LIN {X 0,Y 524.176,Z 655.147,A -85,B 0,C 180,E1 -4756.825,E2 -4756.825} C_VEL
LIN {X 0,Y 523.934,Z 664.266,A -85,B 0,C 180,E1 -4758.392,E2 -4758.392} C_VEL
LIN {X 0,Y 523.658,Z 671.855,A -85,B 0,C 180,E1 -4759.952,E2 -4759.952} C_VEL
LIN {X 0,Y 523.503,Z 679.465,A -85,B 0,C 180,E1 -4761.897,E2 -4761.897} C_VEL
LIN {X 0,Y 523.41,Z 685.25,A -85,B 0,C 180,E1 -4763.834,E2 -4763.834} C_VEL
LIN {X 0,Y 523.312,Z 688.633,A -85,B 0,C 180,E1 -4765.378,E2 -4765.378} C_VEL
LIN {X 0,Y 523.353,Z 691.091,A -85,B 0,C 180,E1 -4766.921,E2 -4766.921} C_VEL
LIN {X 0,Y 523.268,Z 692.478,A -85,B 0,C 180,E1 -4768.461,E2 -4768.461} C_VEL
LIN {X 0,Y 523.242,Z 693,A -85,B 0,C 180,E1 -4770,E2 -4770} C_VEL
LIN {X 0,Y 523.268,Z 692.477,A -85,B 0,C 180,E1 -4771.539,E2 -4771.539} C_VEL
LIN {X 0,Y 523.353,Z 691.089,A -85,B 0,C 180,E1 -4773.079,E2 -4773.079} C_VEL
LIN {X 0,Y 523.312,Z 688.633,A -85,B 0,C 180,E1 -4774.622,E2 -4774.622} C_VEL
LIN {X 0,Y 523.41,Z 685.253,A -85,B 0,C 180,E1 -4776.167,E2 -4776.167} C_VEL
LIN {X 0,Y 523.503,Z 679.467,A -85,B 0,C 180,E1 -4778.104,E2 -4778.104} C_VEL
LIN {X 0,Y 523.658,Z 671.854,A -85,B 0,C 180,E1 -4780.048,E2 -4780.048} C_VEL
LIN {X 0,Y 523.956,Z 663.711,A -85,B 0,C 180,E1 -4781.715,E2 -4781.715} C_VEL
LIN {X 0,Y 524.176,Z 655.145,A -85,B 0,C 180,E1 -4783.175,E2 -4783.175} C_VEL
LIN {X 0,Y 524.649,Z 644.262,A -85,B 0,C 180,E1 -4784.745,E2 -4784.745} C_VEL
LIN {X 0,Y 525.099,Z 633.027,A -85,B 0,C 180,E1 -4786.124,E2 -4786.124} C_VEL
LIN {X 0,Y 525.666,Z 620.786,A -85,B 0,C 180,E1 -4787.406,E2 -4787.406} C_VEL
LIN {X 0,Y 526.239,Z 607.333,A -85,B 0,C 180,E1 -4788.601,E2 -4788.601} C_VEL
LIN {X 0,Y 526.827,Z 594.297,A -85,B 0,C 180,E1 -4789.583,E2 -4789.583} C_VEL
LIN {X 0,Y 527.381,Z 580.397,A -85,B 0,C 180,E1 -4790.476,E2 -4790.476} C_VEL
LIN {X 0,Y 528.118,Z 564.128,A -85,B 0,C 180,E1 -4791.326,E2 -4791.326} C_VEL
LIN {X 0,Y 528.555,Z 550.131,A -85,B 0,C 180,E1 -4791.909,E2 -4791.909} C_VEL
LIN {X 0,Y 529.007,Z 533.263,A -85,B 0,C 180,E1 -4792.455,E2 -4792.455} C_VEL
LIN {X 0,Y 529.386,Z 516.858,A -85,B 0,C 180,E1 -4792.824,E2 -4792.824} C_VEL
LIN {X 0,Y 530.879,Z 326.095,A -85,B 0,C 180,E1 -4795.547,E2 -4795.547} C_VEL
LIN {X 0,Y 528.167,Z 310.802,A -85,B 0,C 180,E1 -4795.922,E2 -4795.922} C_VEL
LIN {X 0,Y 529.041,Z 286.938,A -85,B 0,C 180,E1 -4798.168,E2 -4798.168} C_VEL
LIN {X 0,Y 523.929,Z 269.536,A -85,B 0,C 180,E1 -4800.201,E2 -4800.201} C_VEL
LIN {X 0,Y 523.94,Z 269.535,A -85,B 0,C 180,E1 -4803.365,E2 -4803.365} C_VEL
LIN {X 0,Y 523.902,Z 269.536,A -85,B 0,C 180,E1 -4806.402,E2 -4806.402} C_VEL
LIN {X 0,Y 523.922,Z 269.536,A -85,B 0,C 180,E1 -4809.085,E2 -4809.085} C_VEL
LIN {X 0,Y 523.957,Z 269.524,A -85,B 0,C 180,E1 -4812.119,E2 -4812.119} C_VEL
LIN {X 0,Y 523.956,Z 269.53,A -85,B 0,C 180,E1 -4815.309,E2 -4815.309} C_VEL
LIN {X 0,Y 523.962,Z 269.527,A -85,B 0,C 180,E1 -4818.689,E2 -4818.689} C_VEL
LIN {X 0,Y 523.917,Z 269.529,A -85,B 0,C 180,E1 -4821.899,E2 -4821.899} C_VEL
LIN {X 0,Y 523.925,Z 269.539,A -85,B 0,C 180,E1 -4824.911,E2 -4824.911} C_VEL
LIN {X 0,Y 523.936,Z 269.527,A -85,B 0,C 180,E1 -4827.68,E2 -4827.68} C_VEL
LIN {X 0,Y 523.955,Z 269.532,A -85,B 0,C 180,E1 -4830.677,E2 -4830.677} C_VEL
LIN {X 0,Y 523.975,Z 269.524,A -85,B 0,C 180,E1 -4833.729,E2 -4833.729} C_VEL
LIN {X 0,Y 523.937,Z 269.53,A -85,B 0,C 180,E1 -4836.271,E2 -4836.271} C_VEL
LIN {X 0,Y 523.947,Z 269.531,A -85,B 0,C 180,E1 -4838.767,E2 -4838.767} C_VEL
LIN {X 0,Y 523.95,Z 269.528,A -85,B 0,C 180,E1 -4841.221,E2 -4841.221} C_VEL
LIN {X 0,Y 523.932,Z 269.522,A -85,B 0,C 180,E1 -4843.639,E2 -4843.639} C_VEL
LIN {X 0,Y 523.934,Z 269.531,A -85,B 0,C 180,E1 -4846.028,E2 -4846.028} C_VEL
LIN {X 0,Y 524.015,Z 269.521,A -85,B 0,C 180,E1 -4848.395,E2 -4848.395} C_VEL
LIN {X 0,Y 523.988,Z 269.522,A -85,B 0,C 180,E1 -4851.516,E2 -4851.516} C_VEL
LIN {X 0,Y 524.069,Z 269.511,A -85,B 0,C 180,E1 -4854.614,E2 -4854.614} C_VEL
LIN {X 0,Y 524.111,Z 269.506,A -85,B 0,C 180,E1 -4857.695,E2 -4857.695} C_VEL
LIN {X 0,Y 524.121,Z 269.503,A -85,B 0,C 180,E1 -4860.769,E2 -4860.769} C_VEL
LIN {X 0,Y 524.006,Z 269.519,A -85,B 0,C 180,E1 -4863.076,E2 -4863.076} C_VEL
LIN {X 0,Y 524.066,Z 269.513,A -85,B 0,C 180,E1 -4865.387,E2 -4865.387} C_VEL
LIN {X 0,Y 523.957,Z 269.526,A -85,B 0,C 180,E1 -4868.485,E2 -4868.485} C_VEL
LIN {X 0,Y 524.002,Z 269.523,A -85,B 0,C 180,E1 -4871.737,E2 -4871.737} C_VEL
LIN {X 0,Y 523.99,Z 269.521,A -85,B 0,C 180,E1 -4875.05,E2 -4875.05} C_VEL
LIN {X 0,Y 523.917,Z 269.537,A -85,B 0,C 180,E1 -4877.971,E2 -4877.971} C_VEL
LIN {X 0,Y 523.952,Z 269.533,A -85,B 0,C 180,E1 -4880.411,E2 -4880.411} C_VEL
LIN {X 0,Y 523.903,Z 269.531,A -85,B 0,C 180,E1 -4882.894,E2 -4882.894} C_VEL
LIN {X 0,Y 523.879,Z 269.536,A -85,B 0,C 180,E1 -4885.423,E2 -4885.423} C_VEL
LIN {X 0,Y 523.897,Z 269.536,A -85,B 0,C 180,E1 -4888.004,E2 -4888.004} C_VEL
LIN {X 0,Y 523.901,Z 269.534,A -85,B 0,C 180,E1 -4890.846,E2 -4890.846} C_VEL
LIN {X 0,Y 523.914,Z 269.538,A -85,B 0,C 180,E1 -4893.727,E2 -4893.727} C_VEL
LIN {X 0,Y 523.85,Z 269.546,A -85,B 0,C 180,E1 -4896.393,E2 -4896.393} C_VEL
LIN {X 0,Y 523.894,Z 269.535,A -85,B 0,C 180,E1 -4899.088,E2 -4899.088} C_VEL
LIN {X 0,Y 523.889,Z 269.542,A -85,B 0,C 180,E1 -4902.126,E2 -4902.126} C_VEL
LIN {X 0,Y 523.935,Z 269.533,A -85,B 0,C 180,E1 -4905.312,E2 -4905.312} C_VEL
LIN {X 0,Y 523.878,Z 269.537,A -85,B 0,C 180,E1 -4906.903,E2 -4906.903} C_VEL
LIN {X 0,Y 523.085,Z 269.695,A -85,B 0,C 180,E1 -4907.359,E2 -4907.359} C_VEL
LIN {X 0,Y 517.322,Z 270.465,A -85,B 0,C 180,E1 -4908.74,E2 -4908.74} C_VEL
LIN {X 0,Y 517.059,Z 271.408,A -85,B 0,C 180,E1 -4909.06,E2 -4909.06} C_VEL
LIN {X 0,Y 517.156,Z 271.75,A -85,B 0,C 180,E1 -4909.114,E2 -4909.114} C_VEL
LIN {X 0,Y 520.813,Z 284.323,A -85,B 0,C 180,E1 -4910.753,E2 -4910.753} C_VEL
LIN {X 0,Y 522.606,Z 289.121,A -85,B 0,C 180,E1 -4910.923,E2 -4910.923} C_VEL
LIN {X 0,Y 524.602,Z 299.005,A -85,B 0,C 180,E1 -4911.178,E2 -4911.178} C_VEL
LIN {X 0,Y 522.859,Z 490.272,A -85,B 0,C 180,E1 -4913.95,E2 -4913.95} C_VEL
LIN {X 0,Y 522.455,Z 507.382,A -85,B 0,C 180,E1 -4914.364,E2 -4914.364} C_VEL
LIN {X 0,Y 521.966,Z 523.592,A -85,B 0,C 180,E1 -4914.92,E2 -4914.92} C_VEL
LIN {X 0,Y 521.376,Z 539.542,A -85,B 0,C 180,E1 -4915.635,E2 -4915.635} C_VEL
LIN {X 0,Y 520.708,Z 554.605,A -85,B 0,C 180,E1 -4916.475,E2 -4916.475} C_VEL
LIN {X 0,Y 520.002,Z 569.721,A -85,B 0,C 180,E1 -4917.504,E2 -4917.504} C_VEL
LIN {X 0,Y 519.333,Z 583.007,A -85,B 0,C 180,E1 -4918.59,E2 -4918.59} C_VEL
LIN {X 0,Y 518.659,Z 595.537,A -85,B 0,C 180,E1 -4919.797,E2 -4919.797} C_VEL
LIN {X 0,Y 518.053,Z 607.991,A -85,B 0,C 180,E1 -4921.21,E2 -4921.21} C_VEL
LIN {X 0,Y 517.516,Z 619.257,A -85,B 0,C 180,E1 -4922.72,E2 -4922.72} C_VEL
LIN {X 0,Y 517.107,Z 628.765,A -85,B 0,C 180,E1 -4924.22,E2 -4924.22} C_VEL
LIN {X 0,Y 516.772,Z 637.779,A -85,B 0,C 180,E1 -4925.921,E2 -4925.921} C_VEL
LIN {X 0,Y 516.508,Z 645.511,A -85,B 0,C 180,E1 -4927.709,E2 -4927.709} C_VEL
LIN {X 0,Y 516.4,Z 650.992,A -85,B 0,C 180,E1 -4929.277,E2 -4929.277} C_VEL
LIN {X 0,Y 516.251,Z 655.643,A -85,B 0,C 180,E1 -4930.93,E2 -4930.93} C_VEL
LIN {X 0,Y 516.21,Z 659.042,A -85,B 0,C 180,E1 -4932.571,E2 -4932.571} C_VEL
LIN {X 0,Y 516.137,Z 661.375,A -85,B 0,C 180,E1 -4934.197,E2 -4934.197} C_VEL
LIN {X 0,Y 516.177,Z 662.678,A -85,B 0,C 180,E1 -4935.813,E2 -4935.813} C_VEL
LIN {X 0,Y 516.178,Z 662.93,A -85,B 0,C 180,E1 -4937.417,E2 -4937.417} C_VEL
LIN {X 0,Y 516.258,Z 662.227,A -85,B 0,C 180,E1 -4939.013,E2 -4939.013} C_VEL
LIN {X 0,Y 516.163,Z 660.484,A -85,B 0,C 180,E1 -4940.596,E2 -4940.596} C_VEL
LIN {X 0,Y 516.227,Z 657.838,A -85,B 0,C 180,E1 -4942.175,E2 -4942.175} C_VEL
LIN {X 0,Y 516.391,Z 653.034,A -85,B 0,C 180,E1 -4944.141,E2 -4944.141} C_VEL
LIN {X 0,Y 516.455,Z 647.983,A -85,B 0,C 180,E1 -4945.708,E2 -4945.708} C_VEL
LIN {X 0,Y 516.589,Z 641.868,A -85,B 0,C 180,E1 -4947.271,E2 -4947.271} C_VEL
LIN {X 0,Y 516.908,Z 633.446,A -85,B 0,C 180,E1 -4949.026,E2 -4949.026} C_VEL
LIN {X 0,Y 517.182,Z 624.422,A -85,B 0,C 180,E1 -4950.584,E2 -4950.584} C_VEL
LIN {X 0,Y 517.716,Z 613.744,A -85,B 0,C 180,E1 -4952.139,E2 -4952.139} C_VEL
LIN {X 0,Y 518.308,Z 602.777,A -85,B 0,C 180,E1 -4953.498,E2 -4953.498} C_VEL
LIN {X 0,Y 518.905,Z 590.953,A -85,B 0,C 180,E1 -4954.758,E2 -4954.758} C_VEL
LIN {X 0,Y 519.574,Z 578.074,A -85,B 0,C 180,E1 -4955.92,E2 -4955.92} C_VEL
LIN {X 0,Y 520.204,Z 564.159,A -85,B 0,C 180,E1 -4956.984,E2 -4956.984} C_VEL
LIN {X 0,Y 520.902,Z 548.964,A -85,B 0,C 180,E1 -4957.949,E2 -4957.949} C_VEL
LIN {X 0,Y 521.584,Z 534.106,A -85,B 0,C 180,E1 -4958.719,E2 -4958.719} C_VEL
LIN {X 0,Y 522.114,Z 519.014,A -85,B 0,C 180,E1 -4959.344,E2 -4959.344} C_VEL
LIN {X 0,Y 522.584,Z 502.822,A -85,B 0,C 180,E1 -4959.849,E2 -4959.849} C_VEL
LIN {X 0,Y 522.925,Z 485.838,A -85,B 0,C 180,E1 -4960.213,E2 -4960.213} C_VEL
LIN {X 0,Y 524.588,Z 299.14,A -85,B 0,C 180,E1 -4962.908,E2 -4962.908} C_VEL
LIN {X 0,Y 521.958,Z 287.007,A -85,B 0,C 180,E1 -4963.232,E2 -4963.232} C_VEL
LIN {X 0,Y 520.663,Z 283.932,A -85,B 0,C 180,E1 -4963.375,E2 -4963.375} C_VEL
LIN {X 0,Y 516.944,Z 270.406,A -85,B 0,C 180,E1 -4965.144,E2 -4965.144} C_VEL
LIN {X 0,Y 516.88,Z 270.415,A -85,B 0,C 180,E1 -4968.224,E2 -4968.224} C_VEL
LIN {X 0,Y 516.903,Z 270.41,A -85,B 0,C 180,E1 -4970.702,E2 -4970.702} C_VEL
LIN {X 0,Y 516.86,Z 270.413,A -85,B 0,C 180,E1 -4973.224,E2 -4973.224} C_VEL
LIN {X 0,Y 516.863,Z 270.412,A -85,B 0,C 180,E1 -4976.177,E2 -4976.177} C_VEL
LIN {X 0,Y 516.906,Z 270.406,A -85,B 0,C 180,E1 -4979.305,E2 -4979.305} C_VEL
LIN {X 0,Y 516.849,Z 270.419,A -85,B 0,C 180,E1 -4982.027,E2 -4982.027} C_VEL
LIN {X 0,Y 516.853,Z 270.41,A -85,B 0,C 180,E1 -4984.827,E2 -4984.827} C_VEL
LIN {X 0,Y 516.828,Z 270.42,A -85,B 0,C 180,E1 -4987.935,E2 -4987.935} C_VEL
LIN {X 0,Y 516.821,Z 270.416,A -85,B 0,C 180,E1 -4990.748,E2 -4990.748} C_VEL
LIN {X 0,Y 516.862,Z 270.417,A -85,B 0,C 180,E1 -4993.905,E2 -4993.905} C_VEL
LIN {X 0,Y 516.861,Z 270.413,A -85,B 0,C 180,E1 -4996.109,E2 -4996.109} C_VEL
LIN {X 0,Y 516.823,Z 270.417,A -85,B 0,C 180,E1 -4999.252,E2 -4999.252} C_VEL
LIN {X 0,Y 516.859,Z 270.402,A -85,B 0,C 180,E1 -5002.06,E2 -5002.06} C_VEL
LIN {X 0,Y 516.871,Z 270.401,A -85,B 0,C 180,E1 -5005.174,E2 -5005.174} C_VEL
LIN {X 0,Y 516.868,Z 270.416,A -85,B 0,C 180,E1 -5007.974,E2 -5007.974} C_VEL
LIN {X 0,Y 516.904,Z 270.4,A -85,B 0,C 180,E1 -5010.694,E2 -5010.694} C_VEL
LIN {X 0,Y 516.879,Z 270.415,A -85,B 0,C 180,E1 -5013.818,E2 -5013.818} C_VEL
LIN {X 0,Y 516.859,Z 270.406,A -85,B 0,C 180,E1 -5016.775,E2 -5016.775} C_VEL
LIN {X 0,Y 516.941,Z 270.407,A -85,B 0,C 180,E1 -5019.731,E2 -5019.731} C_VEL
LIN {X 0,Y 516.895,Z 270.402,A -85,B 0,C 180,E1 -5022.595,E2 -5022.595} C_VEL
LIN {X 0,Y 516.937,Z 270.403,A -85,B 0,C 180,E1 -5025.029,E2 -5025.029} C_VEL
LIN {X 0,Y 516.968,Z 270.393,A -85,B 0,C 180,E1 -5028.233,E2 -5028.233} C_VEL
LIN {X 0,Y 516.952,Z 270.406,A -85,B 0,C 180,E1 -5031.399,E2 -5031.399} C_VEL
LIN {X 0,Y 517.008,Z 270.391,A -85,B 0,C 180,E1 -5033.756,E2 -5033.756} C_VEL
LIN {X 0,Y 517.082,Z 270.388,A -85,B 0,C 180,E1 -5037.663,E2 -5037.663} C_VEL
LIN {X 0,Y 517.091,Z 270.377,A -85,B 0,C 180,E1 -5040.778,E2 -5040.778} C_VEL
LIN {X 0,Y 517.01,Z 270.396,A -85,B 0,C 180,E1 -5043.117,E2 -5043.117} C_VEL
LIN {X 0,Y 516.995,Z 270.388,A -85,B 0,C 180,E1 -5046.243,E2 -5046.243} C_VEL
LIN {X 0,Y 516.968,Z 270.394,A -85,B 0,C 180,E1 -5048.6,E2 -5048.6} C_VEL
LIN {X 0,Y 516.952,Z 270.399,A -85,B 0,C 180,E1 -5051.807,E2 -5051.807} C_VEL
LIN {X 0,Y 516.944,Z 270.408,A -85,B 0,C 180,E1 -5055.146,E2 -5055.146} C_VEL
LIN {X 0,Y 516.916,Z 270.404,A -85,B 0,C 180,E1 -5058.222,E2 -5058.222} C_VEL
LIN {X 0,Y 516.912,Z 270.407,A -85,B 0,C 180,E1 -5060.701,E2 -5060.701} C_VEL
LIN {X 0,Y 516.912,Z 270.405,A -85,B 0,C 180,E1 -5064.072,E2 -5064.072} C_VEL
LIN {X 0,Y 516.924,Z 270.406,A -85,B 0,C 180,E1 -5066.657,E2 -5066.657} C_VEL
LIN {X 0,Y 516.91,Z 270.408,A -85,B 0,C 180,E1 -5069.523,E2 -5069.523} C_VEL
LIN {X 0,Y 516.894,Z 270.409,A -85,B 0,C 180,E1 -5072.543,E2 -5072.543} C_VEL
LIN {X 0,Y 516.878,Z 270.41,A -85,B 0,C 180,E1 -5075.331,E2 -5075.331} C_VEL
LIN {X 0,Y 516.881,Z 270.408,A -85,B 0,C 180,E1 -5077.943,E2 -5077.943} C_VEL
LIN {X 0,Y 516.884,Z 270.412,A -85,B 0,C 180,E1 -5080.741,E2 -5080.741} C_VEL
LIN {X 0,Y 516.902,Z 270.414,A -85,B 0,C 180,E1 -5082.829,E2 -5082.829} C_VEL
LIN {X 0,Y 516.921,Z 270.41,A -85,B 0,C 180,E1 -5085.01,E2 -5085.01} C_VEL
LIN {X 0,Y 516.916,Z 270.406,A -85,B 0,C 180,E1 -5088.398,E2 -5088.398} C_VEL
LIN {X 0,Y 516.881,Z 270.411,A -85,B 0,C 180,E1 -5091.284,E2 -5091.284} C_VEL
LIN {X 0,Y 516.869,Z 270.412,A -85,B 0,C 180,E1 -5094.22,E2 -5094.22} C_VEL
LIN {X 0,Y 516.893,Z 270.413,A -85,B 0,C 180,E1 -5097.053,E2 -5097.053} C_VEL
LIN {X 0,Y 516.929,Z 270.527,A -85,B 0,C 180,E1 -5099.488,E2 -5099.488} C_VEL
LIN {X 0,Y 522.355,Z 288.719,A -85,B 0,C 180,E1 -5101.621,E2 -5101.621} C_VEL
LIN {X 0,Y 521.573,Z 310.709,A -85,B 0,C 180,E1 -5103.726,E2 -5103.726} C_VEL
LIN {X 0,Y 524.448,Z 326.713,A -85,B 0,C 180,E1 -5104.128,E2 -5104.128} C_VEL
LIN {X 0,Y 522.92,Z 512.151,A -85,B 0,C 180,E1 -5106.799,E2 -5106.799} C_VEL
LIN {X 0,Y 522.575,Z 528.492,A -85,B 0,C 180,E1 -5107.123,E2 -5107.123} C_VEL
LIN {X 0,Y 522.146,Z 545.237,A -85,B 0,C 180,E1 -5107.625,E2 -5107.625} C_VEL
LIN {X 0,Y 521.517,Z 560.731,A -85,B 0,C 180,E1 -5108.243,E2 -5108.243} C_VEL
LIN {X 0,Y 520.892,Z 576.679,A -85,B 0,C 180,E1 -5109.051,E2 -5109.051} C_VEL
LIN {X 0,Y 520.318,Z 589.813,A -85,B 0,C 180,E1 -5109.853,E2 -5109.853} C_VEL
LIN {X 0,Y 519.549,Z 604.818,A -85,B 0,C 180,E1 -5110.953,E2 -5110.953} C_VEL
LIN {X 0,Y 518.852,Z 618.478,A -85,B 0,C 180,E1 -5112.154,E2 -5112.154} C_VEL
LIN {X 0,Y 518.225,Z 631.031,A -85,B 0,C 180,E1 -5113.453,E2 -5113.453} C_VEL
LIN {X 0,Y 517.702,Z 642.613,A -85,B 0,C 180,E1 -5114.859,E2 -5114.859} C_VEL
LIN {X 0,Y 517.296,Z 652.447,A -85,B 0,C 180,E1 -5116.246,E2 -5116.246} C_VEL
LIN {X 0,Y 516.945,Z 661.96,A -85,B 0,C 180,E1 -5117.836,E2 -5117.836} C_VEL
LIN {X 0,Y 516.679,Z 669.918,A -85,B 0,C 180,E1 -5119.419,E2 -5119.419} C_VEL
LIN {X 0,Y 516.469,Z 676.56,A -85,B 0,C 180,E1 -5120.997,E2 -5120.997} C_VEL
LIN {X 0,Y 516.388,Z 681.949,A -85,B 0,C 180,E1 -5122.571,E2 -5122.571} C_VEL
LIN {X 0,Y 516.321,Z 685.25,A -85,B 0,C 180,E1 -5123.749,E2 -5123.749} C_VEL
LIN {X 0,Y 516.225,Z 688.633,A -85,B 0,C 180,E1 -5125.315,E2 -5125.315} C_VEL
LIN {X 0,Y 516.267,Z 691.091,A -85,B 0,C 180,E1 -5126.879,E2 -5126.879} C_VEL
LIN {X 0,Y 516.186,Z 692.477,A -85,B 0,C 180,E1 -5128.44,E2 -5128.44} C_VEL
LIN {X 0,Y 516.149,Z 693,A -85,B 0,C 180,E1 -5130,E2 -5130} C_VEL
LIN {X 0,Y 516.186,Z 692.477,A -85,B 0,C 180,E1 -5131.56,E2 -5131.56} C_VEL
LIN {X 0,Y 516.267,Z 691.089,A -85,B 0,C 180,E1 -5133.122,E2 -5133.122} C_VEL
LIN {X 0,Y 516.225,Z 688.632,A -85,B 0,C 180,E1 -5134.686,E2 -5134.686} C_VEL
LIN {X 0,Y 516.368,Z 684.558,A -85,B 0,C 180,E1 -5136.507,E2 -5136.507} C_VEL
LIN {X 0,Y 516.418,Z 679.432,A -85,B 0,C 180,E1 -5138.216,E2 -5138.216} C_VEL
LIN {X 0,Y 516.591,Z 671.737,A -85,B 0,C 180,E1 -5140.187,E2 -5140.187} C_VEL
LIN {X 0,Y 516.933,Z 663.158,A -85,B 0,C 180,E1 -5141.946,E2 -5141.946} C_VEL
LIN {X 0,Y 517.224,Z 653.678,A -85,B 0,C 180,E1 -5143.556,E2 -5143.556} C_VEL
LIN {X 0,Y 517.666,Z 644.035,A -85,B 0,C 180,E1 -5144.949,E2 -5144.949} C_VEL
LIN {X 0,Y 518.146,Z 632.796,A -85,B 0,C 180,E1 -5146.347,E2 -5146.347} C_VEL
LIN {X 0,Y 518.797,Z 620.553,A -85,B 0,C 180,E1 -5147.644,E2 -5147.644} C_VEL
LIN {X 0,Y 519.405,Z 607.56,A -85,B 0,C 180,E1 -5148.814,E2 -5148.814} C_VEL
LIN {X 0,Y 520.077,Z 594.056,A -85,B 0,C 180,E1 -5149.848,E2 -5149.848} C_VEL
LIN {X 0,Y 520.664,Z 580.15,A -85,B 0,C 180,E1 -5150.752,E2 -5150.752} C_VEL
LIN {X 0,Y 521.413,Z 564.912,A -85,B 0,C 180,E1 -5151.561,E2 -5151.561} C_VEL
LIN {X 0,Y 521.947,Z 549.872,A -85,B 0,C 180,E1 -5152.201,E2 -5152.201} C_VEL
LIN {X 0,Y 522.428,Z 532.988,A -85,B 0,C 180,E1 -5152.753,E2 -5152.753} C_VEL
LIN {X 0,Y 522.807,Z 518.057,A -85,B 0,C 180,E1 -5153.102,E2 -5153.102} C_VEL
LIN {X 0,Y 524.294,Z 349.148,A -85,B 0,C 180,E1 -5155.544,E2 -5155.544} C_VEL
LIN {X 0,Y 524.358,Z 326.07,A -85,B 0,C 180,E1 -5155.885,E2 -5155.885} C_VEL
LIN {X 0,Y 521.531,Z 310.656,A -85,B 0,C 180,E1 -5156.27,E2 -5156.27} C_VEL
LIN {X 0,Y 522.322,Z 288.635,A -85,B 0,C 180,E1 -5158.378,E2 -5158.378} C_VEL
LIN {X 0,Y 516.914,Z 270.41,A -85,B 0,C 180,E1 -5160.541,E2 -5160.541} C_VEL
LIN {X 0,Y 516.906,Z 270.409,A -85,B 0,C 180,E1 -5163.88,E2 -5163.88} C_VEL
LIN {X 0,Y 516.876,Z 270.413,A -85,B 0,C 180,E1 -5166.746,E2 -5166.746} C_VEL
LIN {X 0,Y 516.882,Z 270.412,A -85,B 0,C 180,E1 -5169.722,E2 -5169.722} C_VEL
LIN {X 0,Y 516.906,Z 270.406,A -85,B 0,C 180,E1 -5172.761,E2 -5172.761} C_VEL
LIN {X 0,Y 516.922,Z 270.405,A -85,B 0,C 180,E1 -5175.01,E2 -5175.01} C_VEL
LIN {X 0,Y 516.917,Z 270.403,A -85,B 0,C 180,E1 -5178.399,E2 -5178.399} C_VEL
LIN {X 0,Y 516.884,Z 270.41,A -85,B 0,C 180,E1 -5181.285,E2 -5181.285} C_VEL
LIN {X 0,Y 516.871,Z 270.41,A -85,B 0,C 180,E1 -5184.22,E2 -5184.22} C_VEL
LIN {X 0,Y 516.895,Z 270.406,A -85,B 0,C 180,E1 -5187.053,E2 -5187.053} C_VEL
LIN {X 0,Y 516.893,Z 270.407,A -85,B 0,C 180,E1 -5189.797,E2 -5189.797} C_VEL
LIN {X 0,Y 516.927,Z 270.397,A -85,B 0,C 180,E1 -5192.468,E2 -5192.468} C_VEL
LIN {X 0,Y 516.912,Z 270.408,A -85,B 0,C 180,E1 -5195.072,E2 -5195.072} C_VEL
LIN {X 0,Y 516.886,Z 270.405,A -85,B 0,C 180,E1 -5198.463,E2 -5198.463} C_VEL
LIN {X 0,Y 516.903,Z 270.409,A -85,B 0,C 180,E1 -5200.955,E2 -5200.955} C_VEL
LIN {X 0,Y 516.91,Z 270.397,A -85,B 0,C 180,E1 -5203.41,E2 -5203.41} C_VEL
LIN {X 0,Y 516.891,Z 270.407,A -85,B 0,C 180,E1 -5205.834,E2 -5205.834} C_VEL
LIN {X 0,Y 516.951,Z 270.392,A -85,B 0,C 180,E1 -5209.028,E2 -5209.028} C_VEL
LIN {X 0,Y 516.945,Z 270.403,A -85,B 0,C 180,E1 -5212.187,E2 -5212.187} C_VEL
LIN {X 0,Y 517.015,Z 270.39,A -85,B 0,C 180,E1 -5214.54,E2 -5214.54} C_VEL
LIN {X 0,Y 517.082,Z 270.381,A -85,B 0,C 180,E1 -5217.664,E2 -5217.664} C_VEL
LIN {X 0,Y 517.091,Z 270.378,A -85,B 0,C 180,E1 -5220.779,E2 -5220.779} C_VEL
LIN {X 0,Y 516.95,Z 270.397,A -85,B 0,C 180,E1 -5223.118,E2 -5223.118} C_VEL
LIN {X 0,Y 516.975,Z 270.402,A -85,B 0,C 180,E1 -5226.244,E2 -5226.244} C_VEL
LIN {X 0,Y 516.938,Z 270.398,A -85,B 0,C 180,E1 -5229.39,E2 -5229.39} C_VEL
LIN {X 0,Y 516.955,Z 270.402,A -85,B 0,C 180,E1 -5231.807,E2 -5231.807} C_VEL
LIN {X 0,Y 516.942,Z 270.399,A -85,B 0,C 180,E1 -5235.144,E2 -5235.144} C_VEL
LIN {X 0,Y 516.878,Z 270.409,A -85,B 0,C 180,E1 -5238.224,E2 -5238.224} C_VEL
LIN {X 0,Y 516.901,Z 270.408,A -85,B 0,C 180,E1 -5240.702,E2 -5240.702} C_VEL
LIN {X 0,Y 516.855,Z 270.408,A -85,B 0,C 180,E1 -5243.225,E2 -5243.225} C_VEL
LIN {X 0,Y 516.86,Z 270.418,A -85,B 0,C 180,E1 -5246.177,E2 -5246.177} C_VEL
LIN {X 0,Y 516.831,Z 270.415,A -85,B 0,C 180,E1 -5248.421,E2 -5248.421} C_VEL
LIN {X 0,Y 516.85,Z 270.412,A -85,B 0,C 180,E1 -5251.113,E2 -5251.113} C_VEL
LIN {X 0,Y 516.871,Z 270.419,A -85,B 0,C 180,E1 -5253.96,E2 -5253.96} C_VEL
LIN {X 0,Y 516.794,Z 270.422,A -85,B 0,C 180,E1 -5256.754,E2 -5256.754} C_VEL
LIN {X 0,Y 516.828,Z 270.421,A -85,B 0,C 180,E1 -5259.727,E2 -5259.727} C_VEL
LIN {X 0,Y 516.839,Z 270.415,A -85,B 0,C 180,E1 -5262.837,E2 -5262.837} C_VEL
LIN {X 0,Y 516.9,Z 270.408,A -85,B 0,C 180,E1 -5265.007,E2 -5265.007} C_VEL
LIN {X 0,Y 516.835,Z 270.419,A -85,B 0,C 180,E1 -5268.409,E2 -5268.409} C_VEL
LIN {X 0,Y 516.854,Z 270.506,A -85,B 0,C 180,E1 -5268.953,E2 -5268.953} C_VEL
LIN {X 0,Y 517.156,Z 271.75,A -85,B 0,C 180,E1 -5269.114,E2 -5269.114} C_VEL
LIN {X 0,Y 517.325,Z 274.623,A -85,B 0,C 180,E1 -5269.45,E2 -5269.45} C_VEL
LIN {X 0,Y 515.818,Z 279.777,A -85,B 0,C 180,E1 -5269.943,E2 -5269.943} C_VEL
LIN {X 0,Y 514.795,Z 284.168,A -85,B 0,C 180,E1 -5270.269,E2 -5270.269} C_VEL
LIN {X 0,Y 515.055,Z 287.636,A -85,B 0,C 180,E1 -5270.47,E2 -5270.47} C_VEL
LIN {X 0,Y 515.474,Z 288.778,A -85,B 0,C 180,E1 -5270.522,E2 -5270.522} C_VEL
LIN {X 0,Y 516.634,Z 292.231,A -85,B 0,C 180,E1 -5270.64,E2 -5270.64} C_VEL
LIN {X 0,Y 518.213,Z 300.803,A -85,B 0,C 180,E1 -5270.859,E2 -5270.859} C_VEL
LIN {X 0,Y 516.34,Z 490.302,A -85,B 0,C 180,E1 -5273.64,E2 -5273.64} C_VEL
LIN {X 0,Y 515.921,Z 506.884,A -85,B 0,C 180,E1 -5274.041,E2 -5274.041} C_VEL
LIN {X 0,Y 515.432,Z 522.796,A -85,B 0,C 180,E1 -5274.585,E2 -5274.585} C_VEL
LIN {X 0,Y 514.791,Z 539.038,A -85,B 0,C 180,E1 -5275.311,E2 -5275.311} C_VEL
LIN {X 0,Y 514.124,Z 553.479,A -85,B 0,C 180,E1 -5276.112,E2 -5276.112} C_VEL
LIN {X 0,Y 513.387,Z 568.741,A -85,B 0,C 180,E1 -5277.15,E2 -5277.15} C_VEL
LIN {X 0,Y 512.537,Z 583.481,A -85,B 0,C 180,E1 -5278.361,E2 -5278.361} C_VEL
LIN {X 0,Y 511.802,Z 596.206,A -85,B 0,C 180,E1 -5279.609,E2 -5279.609} C_VEL
LIN {X 0,Y 511.137,Z 608.34,A -85,B 0,C 180,E1 -5281.008,E2 -5281.008} C_VEL
LIN {X 0,Y 510.579,Z 619.588,A -85,B 0,C 180,E1 -5282.54,E2 -5282.54} C_VEL
LIN {X 0,Y 510.137,Z 629.076,A -85,B 0,C 180,E1 -5284.061,E2 -5284.061} C_VEL
LIN {X 0,Y 509.741,Z 638.076,A -85,B 0,C 180,E1 -5285.784,E2 -5285.784} C_VEL
LIN {X 0,Y 509.452,Z 645.651,A -85,B 0,C 180,E1 -5287.561,E2 -5287.561} C_VEL
LIN {X 0,Y 509.319,Z 651.91,A -85,B 0,C 180,E1 -5289.399,E2 -5289.399} C_VEL
LIN {X 0,Y 509.215,Z 655.388,A -85,B 0,C 180,E1 -5290.656,E2 -5290.656} C_VEL
LIN {X 0,Y 509.112,Z 658.91,A -85,B 0,C 180,E1 -5292.32,E2 -5292.32} C_VEL
LIN {X 0,Y 509.043,Z 661.39,A -85,B 0,C 180,E1 -5293.971,E2 -5293.971} C_VEL
LIN {X 0,Y 509.09,Z 662.751,A -85,B 0,C 180,E1 -5295.612,E2 -5295.612} C_VEL
LIN {X 0,Y 509.097,Z 663.147,A -85,B 0,C 180,E1 -5297.239,E2 -5297.239} C_VEL
LIN {X 0,Y 509.176,Z 662.521,A -85,B 0,C 180,E1 -5298.858,E2 -5298.858} C_VEL
LIN {X 0,Y 509.074,Z 660.944,A -85,B 0,C 180,E1 -5300.464,E2 -5300.464} C_VEL
LIN {X 0,Y 509.139,Z 658.37,A -85,B 0,C 180,E1 -5302.066,E2 -5302.066} C_VEL
LIN {X 0,Y 509.306,Z 653.717,A -85,B 0,C 180,E1 -5304.06,E2 -5304.06} C_VEL
LIN {X 0,Y 509.375,Z 648.823,A -85,B 0,C 180,E1 -5305.648,E2 -5305.648} C_VEL
LIN {X 0,Y 509.525,Z 642.829,A -85,B 0,C 180,E1 -5307.233,E2 -5307.233} C_VEL
LIN {X 0,Y 509.801,Z 635.532,A -85,B 0,C 180,E1 -5308.815,E2 -5308.815} C_VEL
LIN {X 0,Y 510.131,Z 626.904,A -85,B 0,C 180,E1 -5310.395,E2 -5310.395} C_VEL
LIN {X 0,Y 510.646,Z 616.692,A -85,B 0,C 180,E1 -5311.972,E2 -5311.972} C_VEL
LIN {X 0,Y 511.272,Z 606.158,A -85,B 0,C 180,E1 -5313.349,E2 -5313.349} C_VEL
LIN {X 0,Y 511.939,Z 593.827,A -85,B 0,C 180,E1 -5314.725,E2 -5314.725} C_VEL
LIN {X 0,Y 512.651,Z 580.333,A -85,B 0,C 180,E1 -5316,E2 -5316} C_VEL
LIN {X 0,Y 513.395,Z 566.823,A -85,B 0,C 180,E1 -5317.077,E2 -5317.077} C_VEL
LIN {X 0,Y 514.161,Z 552.191,A -85,B 0,C 180,E1 -5318.054,E2 -5318.054} C_VEL
LIN {X 0,Y 514.902,Z 536.01,A -85,B 0,C 180,E1 -5318.932,E2 -5318.932} C_VEL
LIN {X 0,Y 515.522,Z 519.951,A -85,B 0,C 180,E1 -5319.613,E2 -5319.613} C_VEL
LIN {X 0,Y 516.003,Z 504.073,A -85,B 0,C 180,E1 -5320.124,E2 -5320.124} C_VEL
LIN {X 0,Y 516.383,Z 487.976,A -85,B 0,C 180,E1 -5320.488,E2 -5320.488} C_VEL
LIN {X 0,Y 518.216,Z 300.126,A -85,B 0,C 180,E1 -5323.238,E2 -5323.238} C_VEL
LIN {X 0,Y 516.029,Z 290.06,A -85,B 0,C 180,E1 -5323.512,E2 -5323.512} C_VEL
LIN {X 0,Y 513.492,Z 284.189,A -85,B 0,C 180,E1 -5323.764,E2 -5323.764} C_VEL
LIN {X 0,Y 509.875,Z 271.287,A -85,B 0,C 180,E1 -5325.459,E2 -5325.459} C_VEL
LIN {X 0,Y 509.839,Z 271.292,A -85,B 0,C 180,E1 -5328.484,E2 -5328.484} C_VEL
LIN {X 0,Y 509.846,Z 271.287,A -85,B 0,C 180,E1 -5331.002,E2 -5331.002} C_VEL
LIN {X 0,Y 509.822,Z 271.292,A -85,B 0,C 180,E1 -5333.564,E2 -5333.564} C_VEL
LIN {X 0,Y 509.803,Z 271.292,A -85,B 0,C 180,E1 -5336.352,E2 -5336.352} C_VEL
LIN {X 0,Y 509.836,Z 271.288,A -85,B 0,C 180,E1 -5338.847,E2 -5338.847} C_VEL
LIN {X 0,Y 509.803,Z 271.294,A -85,B 0,C 180,E1 -5341.591,E2 -5341.591} C_VEL
LIN {X 0,Y 509.823,Z 271.289,A -85,B 0,C 180,E1 -5344.416,E2 -5344.416} C_VEL
LIN {X 0,Y 509.753,Z 271.297,A -85,B 0,C 180,E1 -5347.346,E2 -5347.346} C_VEL
LIN {X 0,Y 509.787,Z 271.295,A -85,B 0,C 180,E1 -5350.387,E2 -5350.387} C_VEL
LIN {X 0,Y 509.793,Z 271.293,A -85,B 0,C 180,E1 -5353.575,E2 -5353.575} C_VEL
LIN {X 0,Y 509.792,Z 271.29,A -85,B 0,C 180,E1 -5356.425,E2 -5356.425} C_VEL
LIN {X 0,Y 509.788,Z 271.297,A -85,B 0,C 180,E1 -5359.612,E2 -5359.612} C_VEL
LIN {X 0,Y 509.779,Z 271.277,A -85,B 0,C 180,E1 -5362.655,E2 -5362.655} C_VEL
LIN {X 0,Y 509.84,Z 271.284,A -85,B 0,C 180,E1 -5365.8,E2 -5365.8} C_VEL
LIN {X 0,Y 509.84,Z 271.285,A -85,B 0,C 180,E1 -5368.721,E2 -5368.721} C_VEL
LIN {X 0,Y 509.834,Z 271.282,A -85,B 0,C 180,E1 -5371.153,E2 -5371.153} C_VEL
LIN {X 0,Y 509.848,Z 271.291,A -85,B 0,C 180,E1 -5373.825,E2 -5373.825} C_VEL
LIN {X 0,Y 509.821,Z 271.283,A -85,B 0,C 180,E1 -5376.436,E2 -5376.436} C_VEL
LIN {X 0,Y 509.918,Z 271.28,A -85,B 0,C 180,E1 -5379.844,E2 -5379.844} C_VEL
LIN {X 0,Y 509.863,Z 271.28,A -85,B 0,C 180,E1 -5383.174,E2 -5383.174} C_VEL
LIN {X 0,Y 509.855,Z 271.29,A -85,B 0,C 180,E1 -5385.633,E2 -5385.633} C_VEL
LIN {X 0,Y 509.913,Z 271.272,A -85,B 0,C 180,E1 -5388.874,E2 -5388.874} C_VEL
LIN {X 0,Y 509.92,Z 271.276,A -85,B 0,C 180,E1 -5392.078,E2 -5392.078} C_VEL
LIN {X 0,Y 509.978,Z 271.262,A -85,B 0,C 180,E1 -5394.464,E2 -5394.464} C_VEL
LIN {X 0,Y 510.051,Z 271.264,A -85,B 0,C 180,E1 -5397.63,E2 -5397.63} C_VEL
LIN {X 0,Y 510.057,Z 271.253,A -85,B 0,C 180,E1 -5400,E2 -5400} C_VEL
LIN {X 0,Y 510.055,Z 271.258,A -85,B 0,C 180,E1 -5402.369,E2 -5402.369} C_VEL
LIN {X 0,Y 509.977,Z 271.268,A -85,B 0,C 180,E1 -5405.535,E2 -5405.535} C_VEL
LIN {X 0,Y 509.915,Z 271.273,A -85,B 0,C 180,E1 -5408.72,E2 -5408.72} C_VEL
LIN {X 0,Y 509.905,Z 271.276,A -85,B 0,C 180,E1 -5411.931,E2 -5411.931} C_VEL
LIN {X 0,Y 509.894,Z 271.285,A -85,B 0,C 180,E1 -5415.241,E2 -5415.241} C_VEL
LIN {X 0,Y 509.861,Z 271.284,A -85,B 0,C 180,E1 -5418.483,E2 -5418.483} C_VEL
LIN {X 0,Y 509.85,Z 271.291,A -85,B 0,C 180,E1 -5421.001,E2 -5421.001} C_VEL
LIN {X 0,Y 509.87,Z 271.283,A -85,B 0,C 180,E1 -5424.426,E2 -5424.426} C_VEL
LIN {X 0,Y 509.883,Z 271.289,A -85,B 0,C 180,E1 -5427.055,E2 -5427.055} C_VEL
LIN {X 0,Y 509.856,Z 271.285,A -85,B 0,C 180,E1 -5429.751,E2 -5429.751} C_VEL
LIN {X 0,Y 509.872,Z 271.287,A -85,B 0,C 180,E1 -5432.774,E2 -5432.774} C_VEL
LIN {X 0,Y 509.838,Z 271.285,A -85,B 0,C 180,E1 -5435.58,E2 -5435.58} C_VEL
LIN {X 0,Y 509.85,Z 271.285,A -85,B 0,C 180,E1 -5438.338,E2 -5438.338} C_VEL
LIN {X 0,Y 509.857,Z 271.286,A -85,B 0,C 180,E1 -5441.425,E2 -5441.425} C_VEL
LIN {X 0,Y 509.855,Z 271.287,A -85,B 0,C 180,E1 -5444.668,E2 -5444.668} C_VEL
LIN {X 0,Y 509.86,Z 271.283,A -85,B 0,C 180,E1 -5448.102,E2 -5448.102} C_VEL
LIN {X 0,Y 509.846,Z 271.292,A -85,B 0,C 180,E1 -5450.648,E2 -5450.648} C_VEL
LIN {X 0,Y 509.823,Z 271.289,A -85,B 0,C 180,E1 -5453.647,E2 -5453.647} C_VEL
LIN {X 0,Y 509.857,Z 271.287,A -85,B 0,C 180,E1 -5456.539,E2 -5456.539} C_VEL
LIN {X 0,Y 509.864,Z 271.316,A -85,B 0,C 180,E1 -5459.135,E2 -5459.135} C_VEL
LIN {X 0,Y 515.532,Z 290.23,A -85,B 0,C 180,E1 -5461.385,E2 -5461.385} C_VEL
LIN {X 0,Y 515.619,Z 294.743,A -85,B 0,C 180,E1 -5461.839,E2 -5461.839} C_VEL
LIN {X 0,Y 514.924,Z 310.64,A -85,B 0,C 180,E1 -5463.372,E2 -5463.372} C_VEL
LIN {X 0,Y 518.072,Z 328.616,A -85,B 0,C 180,E1 -5463.817,E2 -5463.817} C_VEL
LIN {X 0,Y 516.286,Z 516.381,A -85,B 0,C 180,E1 -5466.563,E2 -5466.563} C_VEL
LIN {X 0,Y 515.899,Z 532.827,A -85,B 0,C 180,E1 -5466.942,E2 -5466.942} C_VEL
LIN {X 0,Y 515.311,Z 549.714,A -85,B 0,C 180,E1 -5467.497,E2 -5467.497} C_VEL
LIN {X 0,Y 514.714,Z 564.99,A -85,B 0,C 180,E1 -5468.157,E2 -5468.157} C_VEL
LIN {X 0,Y 514.018,Z 579.994,A -85,B 0,C 180,E1 -5468.967,E2 -5468.967} C_VEL
LIN {X 0,Y 513.345,Z 593.889,A -85,B 0,C 180,E1 -5469.881,E2 -5469.881} C_VEL
LIN {X 0,Y 512.601,Z 607.287,A -85,B 0,C 180,E1 -5470.918,E2 -5470.918} C_VEL
LIN {X 0,Y 511.919,Z 620.373,A -85,B 0,C 180,E1 -5472.111,E2 -5472.111} C_VEL
LIN {X 0,Y 511.214,Z 632.608,A -85,B 0,C 180,E1 -5473.425,E2 -5473.425} C_VEL
LIN {X 0,Y 510.687,Z 643.839,A -85,B 0,C 180,E1 -5474.842,E2 -5474.842} C_VEL
LIN {X 0,Y 510.151,Z 654.72,A -85,B 0,C 180,E1 -5476.456,E2 -5476.456} C_VEL
LIN {X 0,Y 509.826,Z 664.357,A -85,B 0,C 180,E1 -5478.163,E2 -5478.163} C_VEL
LIN {X 0,Y 509.538,Z 671.532,A -85,B 0,C 180,E1 -5479.671,E2 -5479.671} C_VEL
LIN {X 0,Y 509.352,Z 679.222,A -85,B 0,C 180,E1 -5481.67,E2 -5481.67} C_VEL
LIN {X 0,Y 509.255,Z 685.072,A -85,B 0,C 180,E1 -5483.661,E2 -5483.661} C_VEL
LIN {X 0,Y 509.142,Z 688.491,A -85,B 0,C 180,E1 -5485.249,E2 -5485.249} C_VEL
LIN {X 0,Y 509.184,Z 690.979,A -85,B 0,C 180,E1 -5486.835,E2 -5486.835} C_VEL
LIN {X 0,Y 509.106,Z 692.38,A -85,B 0,C 180,E1 -5488.418,E2 -5488.418} C_VEL
LIN {X 0,Y 509.061,Z 692.906,A -85,B 0,C 180,E1 -5490,E2 -5490} C_VEL
LIN {X 0,Y 509.106,Z 692.378,A -85,B 0,C 180,E1 -5491.582,E2 -5491.582} C_VEL
LIN {X 0,Y 509.184,Z 690.976,A -85,B 0,C 180,E1 -5493.165,E2 -5493.165} C_VEL
LIN {X 0,Y 509.142,Z 688.488,A -85,B 0,C 180,E1 -5494.751,E2 -5494.751} C_VEL
LIN {X 0,Y 509.264,Z 684.696,A -85,B 0,C 180,E1 -5496.477,E2 -5496.477} C_VEL
LIN {X 0,Y 509.352,Z 679.217,A -85,B 0,C 180,E1 -5498.33,E2 -5498.33} C_VEL
LIN {X 0,Y 509.538,Z 671.519,A -85,B 0,C 180,E1 -5500.33,E2 -5500.33} C_VEL
LIN {X 0,Y 509.873,Z 662.832,A -85,B 0,C 180,E1 -5502.134,E2 -5502.134} C_VEL
LIN {X 0,Y 510.234,Z 653.454,A -85,B 0,C 180,E1 -5503.745,E2 -5503.745} C_VEL
LIN {X 0,Y 510.699,Z 643.808,A -85,B 0,C 180,E1 -5505.157,E2 -5505.157} C_VEL
LIN {X 0,Y 511.213,Z 632.564,A -85,B 0,C 180,E1 -5506.575,E2 -5506.575} C_VEL
LIN {X 0,Y 511.923,Z 620.32,A -85,B 0,C 180,E1 -5507.889,E2 -5507.889} C_VEL
LIN {X 0,Y 512.568,Z 607.748,A -85,B 0,C 180,E1 -5509.037,E2 -5509.037} C_VEL
LIN {X 0,Y 513.328,Z 593.815,A -85,B 0,C 180,E1 -5510.12,E2 -5510.12} C_VEL
LIN {X 0,Y 513.978,Z 579.904,A -85,B 0,C 180,E1 -5511.035,E2 -5511.035} C_VEL
LIN {X 0,Y 514.826,Z 563.691,A -85,B 0,C 180,E1 -5511.901,E2 -5511.901} C_VEL
LIN {X 0,Y 515.399,Z 548.307,A -85,B 0,C 180,E1 -5512.552,E2 -5512.552} C_VEL
LIN {X 0,Y 515.906,Z 531.792,A -85,B 0,C 180,E1 -5513.084,E2 -5513.084} C_VEL
LIN {X 0,Y 516.341,Z 516.237,A -85,B 0,C 180,E1 -5513.435,E2 -5513.435} C_VEL
LIN {X 0,Y 518.06,Z 328.592,A -85,B 0,C 180,E1 -5516.182,E2 -5516.182} C_VEL
LIN {X 0,Y 514.92,Z 310.316,A -85,B 0,C 180,E1 -5516.647,E2 -5516.647} C_VEL
LIN {X 0,Y 515.713,Z 291.348,A -85,B 0,C 180,E1 -5518.488,E2 -5518.488} C_VEL
LIN {X 0,Y 511.386,Z 276.417,A -85,B 0,C 180,E1 -5520.277,E2 -5520.277} C_VEL
LIN {X 0,Y 509.874,Z 271.287,A -85,B 0,C 180,E1 -5520.915,E2 -5520.915} C_VEL
LIN {X 0,Y 509.858,Z 271.29,A -85,B 0,C 180,E1 -5523.461,E2 -5523.461} C_VEL
LIN {X 0,Y 509.824,Z 271.29,A -85,B 0,C 180,E1 -5526.353,E2 -5526.353} C_VEL
LIN {X 0,Y 509.847,Z 271.288,A -85,B 0,C 180,E1 -5529.353,E2 -5529.353} C_VEL
LIN {X 0,Y 509.848,Z 271.282,A -85,B 0,C 180,E1 -5532.489,E2 -5532.489} C_VEL
LIN {X 0,Y 509.857,Z 271.285,A -85,B 0,C 180,E1 -5535.332,E2 -5535.332} C_VEL
LIN {X 0,Y 509.859,Z 271.283,A -85,B 0,C 180,E1 -5538.575,E2 -5538.575} C_VEL
LIN {X 0,Y 509.852,Z 271.281,A -85,B 0,C 180,E1 -5541.787,E2 -5541.787} C_VEL
LIN {X 0,Y 509.83,Z 271.291,A -85,B 0,C 180,E1 -5544.622,E2 -5544.622} C_VEL
LIN {X 0,Y 509.861,Z 271.281,A -85,B 0,C 180,E1 -5547.481,E2 -5547.481} C_VEL
LIN {X 0,Y 509.859,Z 271.284,A -85,B 0,C 180,E1 -5550.274,E2 -5550.274} C_VEL
LIN {X 0,Y 509.884,Z 271.281,A -85,B 0,C 180,E1 -5552.945,E2 -5552.945} C_VEL
LIN {X 0,Y 509.871,Z 271.28,A -85,B 0,C 180,E1 -5555.575,E2 -5555.575} C_VEL
LIN {X 0,Y 509.851,Z 271.289,A -85,B 0,C 180,E1 -5558.999,E2 -5558.999} C_VEL
LIN {X 0,Y 509.883,Z 271.278,A -85,B 0,C 180,E1 -5562.002,E2 -5562.002} C_VEL
LIN {X 0,Y 509.913,Z 271.28,A -85,B 0,C 180,E1 -5564.819,E2 -5564.819} C_VEL
LIN {X 0,Y 509.903,Z 271.277,A -85,B 0,C 180,E1 -5568.125,E2 -5568.125} C_VEL
LIN {X 0,Y 509.904,Z 271.277,A -85,B 0,C 180,E1 -5571.28,E2 -5571.28} C_VEL
LIN {X 0,Y 509.966,Z 271.268,A -85,B 0,C 180,E1 -5574.465,E2 -5574.465} C_VEL
LIN {X 0,Y 510.052,Z 271.257,A -85,B 0,C 180,E1 -5577.631,E2 -5577.631} C_VEL
LIN {X 0,Y 510.041,Z 271.256,A -85,B 0,C 180,E1 -5580.79,E2 -5580.79} C_VEL
LIN {X 0,Y 510.046,Z 271.255,A -85,B 0,C 180,E1 -5582.37,E2 -5582.37} C_VEL
LIN {X 0,Y 509.964,Z 271.27,A -85,B 0,C 180,E1 -5585.536,E2 -5585.536} C_VEL
LIN {X 0,Y 509.887,Z 271.279,A -85,B 0,C 180,E1 -5588.721,E2 -5588.721} C_VEL
LIN {X 0,Y 509.907,Z 271.281,A -85,B 0,C 180,E1 -5591.932,E2 -5591.932} C_VEL
LIN {X 0,Y 509.898,Z 271.276,A -85,B 0,C 180,E1 -5595.242,E2 -5595.242} C_VEL
LIN {X 0,Y 509.837,Z 271.281,A -85,B 0,C 180,E1 -5598.485,E2 -5598.485} C_VEL
LIN {X 0,Y 509.843,Z 271.286,A -85,B 0,C 180,E1 -5601.002,E2 -5601.002} C_VEL
LIN {X 0,Y 509.812,Z 271.287,A -85,B 0,C 180,E1 -5603.565,E2 -5603.565} C_VEL
LIN {X 0,Y 509.801,Z 271.295,A -85,B 0,C 180,E1 -5606.353,E2 -5606.353} C_VEL
LIN {X 0,Y 509.795,Z 271.29,A -85,B 0,C 180,E1 -5608.85,E2 -5608.85} C_VEL
LIN {X 0,Y 509.79,Z 271.295,A -85,B 0,C 180,E1 -5611.593,E2 -5611.593} C_VEL
LIN {X 0,Y 509.823,Z 271.29,A -85,B 0,C 180,E1 -5614.416,E2 -5614.416} C_VEL
LIN {X 0,Y 509.762,Z 271.3,A -85,B 0,C 180,E1 -5617.346,E2 -5617.346} C_VEL
LIN {X 0,Y 509.788,Z 271.294,A -85,B 0,C 180,E1 -5620.388,E2 -5620.388} C_VEL
LIN {X 0,Y 509.794,Z 271.298,A -85,B 0,C 180,E1 -5623.575,E2 -5623.575} C_VEL
LIN {X 0,Y 509.795,Z 271.293,A -85,B 0,C 180,E1 -5626.425,E2 -5626.425} C_VEL
LIN {X 0,Y 509.809,Z 271.464,A -85,B 0,C 180,E1 -5628.601,E2 -5628.601} C_VEL
LIN {X 0,Y 513.677,Z 284.724,A -85,B 0,C 180,E1 -5630.357,E2 -5630.357} C_VEL
LIN {X 0,Y 515.474,Z 288.778,A -85,B 0,C 180,E1 -5630.522,E2 -5630.522} C_VEL
LIN {X 0,Y 516.482,Z 292.352,A -85,B 0,C 180,E1 -5630.633,E2 -5630.633} C_VEL
LIN {X 0,Y 516.424,Z 298.158,A -85,B 0,C 180,E1 -5630.719,E2 -5630.719} C_VEL
LIN {X 0,Y 515.209,Z 304.004,A -85,B 0,C 180,E1 -5630.741,E2 -5630.741} C_VEL
LIN {X 0,Y 512.924,Z 312.093,A -85,B 0,C 180,E1 -5630.737,E2 -5630.737} C_VEL
LIN {X 0,Y 511.8,Z 318.227,A -85,B 0,C 180,E1 -5630.768,E2 -5630.768} C_VEL
LIN {X 0,Y 511.696,Z 320.29,A -85,B 0,C 180,E1 -5630.794,E2 -5630.794} C_VEL
LIN {X 0,Y 509.849,Z 490.743,A -85,B 0,C 180,E1 -5633.329,E2 -5633.329} C_VEL
LIN {X 0,Y 509.39,Z 507.707,A -85,B 0,C 180,E1 -5633.749,E2 -5633.749} C_VEL
LIN {X 0,Y 508.859,Z 523.494,A -85,B 0,C 180,E1 -5634.301,E2 -5634.301} C_VEL
LIN {X 0,Y 508.139,Z 539.966,A -85,B 0,C 180,E1 -5635.052,E2 -5635.052} C_VEL
LIN {X 0,Y 507.42,Z 554.517,A -85,B 0,C 180,E1 -5635.879,E2 -5635.879} C_VEL
LIN {X 0,Y 506.667,Z 569.203,A -85,B 0,C 180,E1 -5636.895,E2 -5636.895} C_VEL
LIN {X 0,Y 505.8,Z 583.086,A -85,B 0,C 180,E1 -5638.049,E2 -5638.049} C_VEL
LIN {X 0,Y 505.052,Z 594.935,A -85,B 0,C 180,E1 -5639.209,E2 -5639.209} C_VEL
LIN {X 0,Y 504.339,Z 606.938,A -85,B 0,C 180,E1 -5640.58,E2 -5640.58} C_VEL
LIN {X 0,Y 503.786,Z 616.942,A -85,B 0,C 180,E1 -5641.912,E2 -5641.912} C_VEL
LIN {X 0,Y 503.25,Z 626.816,A -85,B 0,C 180,E1 -5643.456,E2 -5643.456} C_VEL
LIN {X 0,Y 502.851,Z 635.171,A -85,B 0,C 180,E1 -5644.989,E2 -5644.989} C_VEL
LIN {X 0,Y 502.563,Z 642.209,A -85,B 0,C 180,E1 -5646.512,E2 -5646.512} C_VEL
LIN {X 0,Y 502.329,Z 648.758,A -85,B 0,C 180,E1 -5648.238,E2 -5648.238} C_VEL
LIN {X 0,Y 502.248,Z 653.182,A -85,B 0,C 180,E1 -5649.643,E2 -5649.643} C_VEL
LIN {X 0,Y 502.082,Z 657.073,A -85,B 0,C 180,E1 -5651.219,E2 -5651.219} C_VEL
LIN {X 0,Y 502.01,Z 660.222,A -85,B 0,C 180,E1 -5652.903,E2 -5652.903} C_VEL
LIN {X 0,Y 501.945,Z 662.232,A -85,B 0,C 180,E1 -5654.572,E2 -5654.572} C_VEL
LIN {X 0,Y 501.993,Z 663.233,A -85,B 0,C 180,E1 -5656.231,E2 -5656.231} C_VEL
LIN {X 0,Y 502.024,Z 663.228,A -85,B 0,C 180,E1 -5657.878,E2 -5657.878} C_VEL
LIN {X 0,Y 502.033,Z 662.23,A -85,B 0,C 180,E1 -5659.514,E2 -5659.514} C_VEL
LIN {X 0,Y 502.027,Z 660.279,A -85,B 0,C 180,E1 -5661.142,E2 -5661.142} C_VEL
LIN {X 0,Y 502.109,Z 657.296,A -85,B 0,C 180,E1 -5662.763,E2 -5662.763} C_VEL
LIN {X 0,Y 502.257,Z 653.344,A -85,B 0,C 180,E1 -5664.379,E2 -5664.379} C_VEL
LIN {X 0,Y 502.381,Z 646.865,A -85,B 0,C 180,E1 -5666.391,E2 -5666.391} C_VEL
LIN {X 0,Y 502.584,Z 640.345,A -85,B 0,C 180,E1 -5667.996,E2 -5667.996} C_VEL
LIN {X 0,Y 503.012,Z 631.494,A -85,B 0,C 180,E1 -5669.8,E2 -5669.8} C_VEL
LIN {X 0,Y 503.406,Z 622.101,A -85,B 0,C 180,E1 -5671.4,E2 -5671.4} C_VEL
LIN {X 0,Y 504.129,Z 610.935,A -85,B 0,C 180,E1 -5672.997,E2 -5672.997} C_VEL
LIN {X 0,Y 504.81,Z 599.42,A -85,B 0,C 180,E1 -5674.391,E2 -5674.391} C_VEL
LIN {X 0,Y 505.531,Z 586.856,A -85,B 0,C 180,E1 -5675.685,E2 -5675.685} C_VEL
LIN {X 0,Y 506.294,Z 573.212,A -85,B 0,C 180,E1 -5676.876,E2 -5676.876} C_VEL
LIN {X 0,Y 507.138,Z 558.26,A -85,B 0,C 180,E1 -5677.966,E2 -5677.966} C_VEL
LIN {X 0,Y 507.941,Z 543.465,A -85,B 0,C 180,E1 -5678.855,E2 -5678.855} C_VEL
LIN {X 0,Y 508.651,Z 528.229,A -85,B 0,C 180,E1 -5679.594,E2 -5679.594} C_VEL
LIN {X 0,Y 509.234,Z 512.555,A -85,B 0,C 180,E1 -5680.185,E2 -5680.185} C_VEL
LIN {X 0,Y 509.663,Z 496.742,A -85,B 0,C 180,E1 -5680.628,E2 -5680.628} C_VEL
LIN {X 0,Y 510.037,Z 479.377,A -85,B 0,C 180,E1 -5680.947,E2 -5680.947} C_VEL
LIN {X 0,Y 511.854,Z 301.541,A -85,B 0,C 180,E1 -5683.568,E2 -5683.568} C_VEL
LIN {X 0,Y 509.902,Z 292.596,A -85,B 0,C 180,E1 -5683.816,E2 -5683.816} C_VEL
LIN {X 0,Y 506.314,Z 284.481,A -85,B 0,C 180,E1 -5684.159,E2 -5684.159} C_VEL
LIN {X 0,Y 502.803,Z 272.168,A -85,B 0,C 180,E1 -5685.804,E2 -5685.804} C_VEL
LIN {X 0,Y 502.812,Z 272.167,A -85,B 0,C 180,E1 -5688.752,E2 -5688.752} C_VEL
LIN {X 0,Y 502.782,Z 272.166,A -85,B 0,C 180,E1 -5691.311,E2 -5691.311} C_VEL
LIN {X 0,Y 502.77,Z 272.174,A -85,B 0,C 180,E1 -5693.915,E2 -5693.915} C_VEL
LIN {X 0,Y 502.76,Z 272.171,A -85,B 0,C 180,E1 -5696.572,E2 -5696.572} C_VEL
LIN {X 0,Y 502.794,Z 272.165,A -85,B 0,C 180,E1 -5699.29,E2 -5699.29} C_VEL
LIN {X 0,Y 502.764,Z 272.173,A -85,B 0,C 180,E1 -5702.086,E2 -5702.086} C_VEL
LIN {X 0,Y 502.752,Z 272.166,A -85,B 0,C 180,E1 -5704.969,E2 -5704.969} C_VEL
LIN {X 0,Y 502.745,Z 272.171,A -85,B 0,C 180,E1 -5708.478,E2 -5708.478} C_VEL
LIN {X 0,Y 502.751,Z 272.168,A -85,B 0,C 180,E1 -5711.073,E2 -5711.073} C_VEL
LIN {X 0,Y 502.78,Z 272.166,A -85,B 0,C 180,E1 -5714.529,E2 -5714.529} C_VEL
LIN {X 0,Y 502.736,Z 272.174,A -85,B 0,C 180,E1 -5717.854,E2 -5717.854} C_VEL
LIN {X 0,Y 502.777,Z 272.161,A -85,B 0,C 180,E1 -5721.021,E2 -5721.021} C_VEL
LIN {X 0,Y 502.751,Z 272.159,A -85,B 0,C 180,E1 -5724.173,E2 -5724.173} C_VEL
LIN {X 0,Y 502.804,Z 272.16,A -85,B 0,C 180,E1 -5726.998,E2 -5726.998} C_VEL
LIN {X 0,Y 502.811,Z 272.159,A -85,B 0,C 180,E1 -5730.066,E2 -5730.066} C_VEL
LIN {X 0,Y 502.775,Z 272.17,A -85,B 0,C 180,E1 -5733.46,E2 -5733.46} C_VEL
LIN {X 0,Y 502.768,Z 272.164,A -85,B 0,C 180,E1 -5736.085,E2 -5736.085} C_VEL
LIN {X 0,Y 502.785,Z 272.164,A -85,B 0,C 180,E1 -5738.688,E2 -5738.688} C_VEL
LIN {X 0,Y 502.824,Z 272.161,A -85,B 0,C 180,E1 -5741.248,E2 -5741.248} C_VEL
LIN {X 0,Y 502.85,Z 272.156,A -85,B 0,C 180,E1 -5744.6,E2 -5744.6} C_VEL
LIN {X 0,Y 502.878,Z 272.149,A -85,B 0,C 180,E1 -5748.039,E2 -5748.039} C_VEL
LIN {X 0,Y 502.862,Z 272.158,A -85,B 0,C 180,E1 -5751.156,E2 -5751.156} C_VEL
LIN {X 0,Y 502.911,Z 272.148,A -85,B 0,C 180,E1 -5753.581,E2 -5753.581} C_VEL
LIN {X 0,Y 502.864,Z 272.155,A -85,B 0,C 180,E1 -5756.795,E2 -5756.795} C_VEL
LIN {X 0,Y 503.033,Z 272.138,A -85,B 0,C 180,E1 -5759.199,E2 -5759.199} C_VEL
LIN {X 0,Y 503.024,Z 272.133,A -85,B 0,C 180,E1 -5762.402,E2 -5762.402} C_VEL
LIN {X 0,Y 502.93,Z 272.144,A -85,B 0,C 180,E1 -5765.613,E2 -5765.613} C_VEL
LIN {X 0,Y 502.873,Z 272.151,A -85,B 0,C 180,E1 -5768.843,E2 -5768.843} C_VEL
LIN {X 0,Y 502.846,Z 272.155,A -85,B 0,C 180,E1 -5772.101,E2 -5772.101} C_VEL
LIN {X 0,Y 502.849,Z 272.161,A -85,B 0,C 180,E1 -5775.399,E2 -5775.399} C_VEL
LIN {X 0,Y 502.826,Z 272.162,A -85,B 0,C 180,E1 -5778.751,E2 -5778.751} C_VEL
LIN {X 0,Y 502.783,Z 272.17,A -85,B 0,C 180,E1 -5781.311,E2 -5781.311} C_VEL
LIN {X 0,Y 502.792,Z 272.165,A -85,B 0,C 180,E1 -5783.913,E2 -5783.913} C_VEL
LIN {X 0,Y 502.863,Z 272.157,A -85,B 0,C 180,E1 -5786.566,E2 -5786.566} C_VEL
LIN {X 0,Y 502.823,Z 272.166,A -85,B 0,C 180,E1 -5789.287,E2 -5789.287} C_VEL
LIN {X 0,Y 502.782,Z 272.165,A -85,B 0,C 180,E1 -5792.084,E2 -5792.084} C_VEL
LIN {X 0,Y 502.806,Z 272.169,A -85,B 0,C 180,E1 -5794.965,E2 -5794.965} C_VEL
LIN {X 0,Y 502.793,Z 272.163,A -85,B 0,C 180,E1 -5797.953,E2 -5797.953} C_VEL
LIN {X 0,Y 502.819,Z 272.163,A -85,B 0,C 180,E1 -5801.065,E2 -5801.065} C_VEL
LIN {X 0,Y 502.789,Z 272.165,A -85,B 0,C 180,E1 -5804.338,E2 -5804.338} C_VEL
LIN {X 0,Y 502.785,Z 272.17,A -85,B 0,C 180,E1 -5806.77,E2 -5806.77} C_VEL
LIN {X 0,Y 502.818,Z 272.167,A -85,B 0,C 180,E1 -5809.005,E2 -5809.005} C_VEL
LIN {X 0,Y 502.792,Z 272.164,A -85,B 0,C 180,E1 -5812.046,E2 -5812.046} C_VEL
LIN {X 0,Y 502.797,Z 272.168,A -85,B 0,C 180,E1 -5815.034,E2 -5815.034} C_VEL
LIN {X 0,Y 502.781,Z 272.169,A -85,B 0,C 180,E1 -5817.915,E2 -5817.915} C_VEL
LIN {X 0,Y 502.841,Z 272.249,A -85,B 0,C 180,E1 -5818.793,E2 -5818.793} C_VEL
LIN {X 0,Y 508.813,Z 292.239,A -85,B 0,C 180,E1 -5821.203,E2 -5821.203} C_VEL
LIN {X 0,Y 509.041,Z 294.486,A -85,B 0,C 180,E1 -5821.442,E2 -5821.442} C_VEL
LIN {X 0,Y 508.297,Z 310.296,A -85,B 0,C 180,E1 -5822.987,E2 -5822.987} C_VEL
LIN {X 0,Y 511.702,Z 329.335,A -85,B 0,C 180,E1 -5823.482,E2 -5823.482} C_VEL
LIN {X 0,Y 509.763,Z 516.092,A -85,B 0,C 180,E1 -5826.245,E2 -5826.245} C_VEL
LIN {X 0,Y 509.342,Z 532.57,A -85,B 0,C 180,E1 -5826.628,E2 -5826.628} C_VEL
LIN {X 0,Y 508.74,Z 549.472,A -85,B 0,C 180,E1 -5827.19,E2 -5827.19} C_VEL
LIN {X 0,Y 508.083,Z 564.756,A -85,B 0,C 180,E1 -5827.857,E2 -5827.857} C_VEL
LIN {X 0,Y 507.34,Z 579.943,A -85,B 0,C 180,E1 -5828.687,E2 -5828.687} C_VEL
LIN {X 0,Y 506.611,Z 593.664,A -85,B 0,C 180,E1 -5829.602,E2 -5829.602} C_VEL
LIN {X 0,Y 505.816,Z 606.818,A -85,B 0,C 180,E1 -5830.63,E2 -5830.63} C_VEL
LIN {X 0,Y 505.042,Z 620.153,A -85,B 0,C 180,E1 -5831.859,E2 -5831.859} C_VEL
LIN {X 0,Y 504.296,Z 632.39,A -85,B 0,C 180,E1 -5833.191,E2 -5833.191} C_VEL
LIN {X 0,Y 503.717,Z 643.624,A -85,B 0,C 180,E1 -5834.628,E2 -5834.628} C_VEL
LIN {X 0,Y 503.172,Z 654.508,A -85,B 0,C 180,E1 -5836.264,E2 -5836.264} C_VEL
LIN {X 0,Y 502.794,Z 663.658,A -85,B 0,C 180,E1 -5837.897,E2 -5837.897} C_VEL
LIN {X 0,Y 502.493,Z 671.322,A -85,B 0,C 180,E1 -5839.524,E2 -5839.524} C_VEL
LIN {X 0,Y 502.256,Z 679.013,A -85,B 0,C 180,E1 -5841.551,E2 -5841.551} C_VEL
LIN {X 0,Y 502.182,Z 684.865,A -85,B 0,C 180,E1 -5843.572,E2 -5843.572} C_VEL
LIN {X 0,Y 502.061,Z 688.284,A -85,B 0,C 180,E1 -5845.182,E2 -5845.182} C_VEL
LIN {X 0,Y 502.102,Z 690.773,A -85,B 0,C 180,E1 -5846.791,E2 -5846.791} C_VEL
LIN {X 0,Y 502.029,Z 692.174,A -85,B 0,C 180,E1 -5848.396,E2 -5848.396} C_VEL
LIN {X 0,Y 501.975,Z 692.7,A -85,B 0,C 180,E1 -5850,E2 -5850} C_VEL
LIN {X 0,Y 502.03,Z 692.171,A -85,B 0,C 180,E1 -5851.604,E2 -5851.604} C_VEL
LIN {X 0,Y 502.102,Z 690.767,A -85,B 0,C 180,E1 -5853.21,E2 -5853.21} C_VEL
LIN {X 0,Y 502.061,Z 688.277,A -85,B 0,C 180,E1 -5854.818,E2 -5854.818} C_VEL
LIN {X 0,Y 502.183,Z 684.749,A -85,B 0,C 180,E1 -5856.469,E2 -5856.469} C_VEL
LIN {X 0,Y 502.256,Z 679.001,A -85,B 0,C 180,E1 -5858.449,E2 -5858.449} C_VEL
LIN {X 0,Y 502.493,Z 671.301,A -85,B 0,C 180,E1 -5860.476,E2 -5860.476} C_VEL
LIN {X 0,Y 502.84,Z 662.611,A -85,B 0,C 180,E1 -5862.307,E2 -5862.307} C_VEL
LIN {X 0,Y 503.225,Z 653.23,A -85,B 0,C 180,E1 -5863.94,E2 -5863.94} C_VEL
LIN {X 0,Y 503.731,Z 643.579,A -85,B 0,C 180,E1 -5865.372,E2 -5865.372} C_VEL
LIN {X 0,Y 504.295,Z 632.333,A -85,B 0,C 180,E1 -5866.809,E2 -5866.809} C_VEL
LIN {X 0,Y 505.03,Z 620.086,A -85,B 0,C 180,E1 -5868.142,E2 -5868.142} C_VEL
LIN {X 0,Y 505.787,Z 606.744,A -85,B 0,C 180,E1 -5869.371,E2 -5869.371} C_VEL
LIN {X 0,Y 506.549,Z 593.571,A -85,B 0,C 180,E1 -5870.401,E2 -5870.401} C_VEL
LIN {X 0,Y 507.298,Z 579.853,A -85,B 0,C 180,E1 -5871.313,E2 -5871.313} C_VEL
LIN {X 0,Y 508.098,Z 565.032,A -85,B 0,C 180,E1 -5872.122,E2 -5872.122} C_VEL
LIN {X 0,Y 508.703,Z 550.652,A -85,B 0,C 180,E1 -5872.758,E2 -5872.758} C_VEL
LIN {X 0,Y 509.277,Z 534.266,A -85,B 0,C 180,E1 -5873.321,E2 -5873.321} C_VEL
LIN {X 0,Y 509.747,Z 518.776,A -85,B 0,C 180,E1 -5873.702,E2 -5873.702} C_VEL
LIN {X 0,Y 510.401,Z 455.201,A -85,B 0,C 180,E1 -5874.662,E2 -5874.662} C_VEL
LIN {X 0,Y 511.666,Z 328.979,A -85,B 0,C 180,E1 -5876.528,E2 -5876.528} C_VEL
LIN {X 0,Y 508.304,Z 310.052,A -85,B 0,C 180,E1 -5877.033,E2 -5877.033} C_VEL
LIN {X 0,Y 509.091,Z 293.464,A -85,B 0,C 180,E1 -5878.668,E2 -5878.668} C_VEL
LIN {X 0,Y 505.059,Z 279.467,A -85,B 0,C 180,E1 -5880.375,E2 -5880.375} C_VEL
LIN {X 0,Y 502.818,Z 272.164,A -85,B 0,C 180,E1 -5881.319,E2 -5881.319} C_VEL
LIN {X 0,Y 502.803,Z 272.166,A -85,B 0,C 180,E1 -5883.994,E2 -5883.994} C_VEL
LIN {X 0,Y 502.777,Z 272.169,A -85,B 0,C 180,E1 -5887.178,E2 -5887.178} C_VEL
LIN {X 0,Y 502.788,Z 272.166,A -85,B 0,C 180,E1 -5890.015,E2 -5890.015} C_VEL
LIN {X 0,Y 502.803,Z 272.158,A -85,B 0,C 180,E1 -5892.2,E2 -5892.2} C_VEL
LIN {X 0,Y 502.801,Z 272.164,A -85,B 0,C 180,E1 -5895.469,E2 -5895.469} C_VEL
LIN {X 0,Y 502.821,Z 272.16,A -85,B 0,C 180,E1 -5898.935,E2 -5898.935} C_VEL
LIN {X 0,Y 502.794,Z 272.16,A -85,B 0,C 180,E1 -5902.047,E2 -5902.047} C_VEL
LIN {X 0,Y 502.799,Z 272.168,A -85,B 0,C 180,E1 -5905.035,E2 -5905.035} C_VEL
LIN {X 0,Y 502.783,Z 272.161,A -85,B 0,C 180,E1 -5907.916,E2 -5907.916} C_VEL
LIN {X 0,Y 502.825,Z 272.161,A -85,B 0,C 180,E1 -5910.713,E2 -5910.713} C_VEL
LIN {X 0,Y 502.864,Z 272.155,A -85,B 0,C 180,E1 -5913.44,E2 -5913.44} C_VEL
LIN {X 0,Y 502.793,Z 272.162,A -85,B 0,C 180,E1 -5916.087,E2 -5916.087} C_VEL
LIN {X 0,Y 502.784,Z 272.164,A -85,B 0,C 180,E1 -5918.689,E2 -5918.689} C_VEL
LIN {X 0,Y 502.831,Z 272.158,A -85,B 0,C 180,E1 -5921.249,E2 -5921.249} C_VEL
LIN {X 0,Y 502.82,Z 272.151,A -85,B 0,C 180,E1 -5923.767,E2 -5923.767} C_VEL
LIN {X 0,Y 502.828,Z 272.162,A -85,B 0,C 180,E1 -5926.255,E2 -5926.255} C_VEL
LIN {X 0,Y 502.878,Z 272.146,A -85,B 0,C 180,E1 -5928.717,E2 -5928.717} C_VEL
LIN {X 0,Y 502.874,Z 272.154,A -85,B 0,C 180,E1 -5931.967,E2 -5931.967} C_VEL
LIN {X 0,Y 502.919,Z 272.147,A -85,B 0,C 180,E1 -5934.387,E2 -5934.387} C_VEL
LIN {X 0,Y 503.021,Z 272.133,A -85,B 0,C 180,E1 -5937.598,E2 -5937.598} C_VEL
LIN {X 0,Y 502.992,Z 272.133,A -85,B 0,C 180,E1 -5940.801,E2 -5940.801} C_VEL
LIN {X 0,Y 503.014,Z 272.13,A -85,B 0,C 180,E1 -5942.403,E2 -5942.403} C_VEL
LIN {X 0,Y 502.917,Z 272.149,A -85,B 0,C 180,E1 -5945.614,E2 -5945.614} C_VEL
LIN {X 0,Y 502.851,Z 272.154,A -85,B 0,C 180,E1 -5948.844,E2 -5948.844} C_VEL
LIN {X 0,Y 502.848,Z 272.162,A -85,B 0,C 180,E1 -5952.102,E2 -5952.102} C_VEL
LIN {X 0,Y 502.849,Z 272.154,A -85,B 0,C 180,E1 -5955.4,E2 -5955.4} C_VEL
LIN {X 0,Y 502.81,Z 272.153,A -85,B 0,C 180,E1 -5958.753,E2 -5958.753} C_VEL
LIN {X 0,Y 502.779,Z 272.166,A -85,B 0,C 180,E1 -5961.312,E2 -5961.312} C_VEL
LIN {X 0,Y 502.758,Z 272.166,A -85,B 0,C 180,E1 -5963.916,E2 -5963.916} C_VEL
LIN {X 0,Y 502.759,Z 272.169,A -85,B 0,C 180,E1 -5966.573,E2 -5966.573} C_VEL
LIN {X 0,Y 502.755,Z 272.167,A -85,B 0,C 180,E1 -5969.293,E2 -5969.293} C_VEL
LIN {X 0,Y 502.758,Z 272.169,A -85,B 0,C 180,E1 -5972.087,E2 -5972.087} C_VEL
LIN {X 0,Y 502.752,Z 272.168,A -85,B 0,C 180,E1 -5974.97,E2 -5974.97} C_VEL
LIN {X 0,Y 502.751,Z 272.17,A -85,B 0,C 180,E1 -5978.48,E2 -5978.48} C_VEL
LIN {X 0,Y 502.752,Z 272.169,A -85,B 0,C 180,E1 -5981.073,E2 -5981.073} C_VEL
LIN {X 0,Y 502.781,Z 272.168,A -85,B 0,C 180,E1 -5984.529,E2 -5984.529} C_VEL
LIN {X 0,Y 502.74,Z 272.175,A -85,B 0,C 180,E1 -5987.855,E2 -5987.855} C_VEL
LIN {X 0,Y 502.759,Z 272.248,A -85,B 0,C 180,E1 -5988.213,E2 -5988.213} C_VEL
LIN {X 0,Y 506.538,Z 285.102,A -85,B 0,C 180,E1 -5989.941,E2 -5989.941} C_VEL
LIN {X 0,Y 510.407,Z 293.94,A -85,B 0,C 180,E1 -5990.31,E2 -5990.31} C_VEL
LIN {X 0,Y 511.864,Z 301.968,A -85,B 0,C 180,E1 -5990.52,E2 -5990.52} C_VEL
LIN {X 0,Y 511.696,Z 320.29,A -85,B 0,C 180,E1 -5990.794,E2 -5990.794} C_VEL
LIN {X 0,Y 511.022,Z 326.153,A -85,B 0,C 180,E1 -5990.847,E2 -5990.847} C_VEL
LIN {X 0,Y 505.56,Z 345.256,A -85,B 0,C 180,E1 -5990.831,E2 -5990.831} C_VEL
LIN {X 0,Y 505.018,Z 351.105,A -85,B 0,C 180,E1 -5990.892,E2 -5990.892} C_VEL
LIN {X 0,Y 503.391,Z 490.352,A -85,B 0,C 180,E1 -5992.993,E2 -5992.993} C_VEL
LIN {X 0,Y 502.887,Z 507.172,A -85,B 0,C 180,E1 -5993.406,E2 -5993.406} C_VEL
LIN {X 0,Y 502.357,Z 522.819,A -85,B 0,C 180,E1 -5993.952,E2 -5993.952} C_VEL
LIN {X 0,Y 501.646,Z 538.611,A -85,B 0,C 180,E1 -5994.666,E2 -5994.666} C_VEL
LIN {X 0,Y 500.87,Z 553.276,A -85,B 0,C 180,E1 -5995.492,E2 -5995.492} C_VEL
LIN {X 0,Y 499.973,Z 568.268,A -85,B 0,C 180,E1 -5996.527,E2 -5996.527} C_VEL
LIN {X 0,Y 499.141,Z 581.829,A -85,B 0,C 180,E1 -5997.653,E2 -5997.653} C_VEL
LIN {X 0,Y 498.308,Z 594.583,A -85,B 0,C 180,E1 -5998.899,E2 -5998.899} C_VEL
LIN {X 0,Y 497.606,Z 605.533,A -85,B 0,C 180,E1 -6000.141,E2 -6000.141} C_VEL
LIN {X 0,Y 496.866,Z 617.283,A -85,B 0,C 180,E1 -6001.716,E2 -6001.716} C_VEL
LIN {X 0,Y 496.303,Z 626.833,A -85,B 0,C 180,E1 -6003.229,E2 -6003.229} C_VEL
LIN {X 0,Y 495.857,Z 635.472,A -85,B 0,C 180,E1 -6004.836,E2 -6004.836} C_VEL
LIN {X 0,Y 495.493,Z 643.394,A -85,B 0,C 180,E1 -6006.6,E2 -6006.6} C_VEL
LIN {X 0,Y 495.254,Z 649.78,A -85,B 0,C 180,E1 -6008.348,E2 -6008.348} C_VEL
LIN {X 0,Y 495.133,Z 654.799,A -85,B 0,C 180,E1 -6010.083,E2 -6010.083} C_VEL
LIN {X 0,Y 494.95,Z 659.105,A -85,B 0,C 180,E1 -6012.058,E2 -6012.058} C_VEL
LIN {X 0,Y 494.881,Z 661.323,A -85,B 0,C 180,E1 -6013.499,E2 -6013.499} C_VEL
LIN {X 0,Y 494.916,Z 662.946,A -85,B 0,C 180,E1 -6015.19,E2 -6015.19} C_VEL
LIN {X 0,Y 494.912,Z 663.565,A -85,B 0,C 180,E1 -6016.867,E2 -6016.867} C_VEL
LIN {X 0,Y 494.993,Z 663.152,A -85,B 0,C 180,E1 -6018.535,E2 -6018.535} C_VEL
LIN {X 0,Y 494.918,Z 661.817,A -85,B 0,C 180,E1 -6020.189,E2 -6020.189} C_VEL
LIN {X 0,Y 494.949,Z 659.437,A -85,B 0,C 180,E1 -6021.837,E2 -6021.837} C_VEL
LIN {X 0,Y 495.113,Z 655.99,A -85,B 0,C 180,E1 -6023.535,E2 -6023.535} C_VEL
LIN {X 0,Y 495.221,Z 650.469,A -85,B 0,C 180,E1 -6025.523,E2 -6025.523} C_VEL
LIN {X 0,Y 495.405,Z 644.67,A -85,B 0,C 180,E1 -6027.154,E2 -6027.154} C_VEL
LIN {X 0,Y 495.704,Z 637.726,A -85,B 0,C 180,E1 -6028.781,E2 -6028.781} C_VEL
LIN {X 0,Y 496.082,Z 629.435,A -85,B 0,C 180,E1 -6030.406,E2 -6030.406} C_VEL
LIN {X 0,Y 496.637,Z 619.554,A -85,B 0,C 180,E1 -6032.027,E2 -6032.027} C_VEL
LIN {X 0,Y 497.352,Z 609.417,A -85,B 0,C 180,E1 -6033.443,E2 -6033.443} C_VEL
LIN {X 0,Y 498.104,Z 597.637,A -85,B 0,C 180,E1 -6034.856,E2 -6034.856} C_VEL
LIN {X 0,Y 498.868,Z 584.81,A -85,B 0,C 180,E1 -6036.167,E2 -6036.167} C_VEL
LIN {X 0,Y 499.792,Z 570.674,A -85,B 0,C 180,E1 -6037.372,E2 -6037.372} C_VEL
LIN {X 0,Y 500.62,Z 556.627,A -85,B 0,C 180,E1 -6038.375,E2 -6038.375} C_VEL
LIN {X 0,Y 501.416,Z 541.398,A -85,B 0,C 180,E1 -6039.276,E2 -6039.276} C_VEL
LIN {X 0,Y 502.16,Z 525.601,A -85,B 0,C 180,E1 -6040.024,E2 -6040.024} C_VEL
LIN {X 0,Y 502.818,Z 509.16,A -85,B 0,C 180,E1 -6040.622,E2 -6040.622} C_VEL
LIN {X 0,Y 503.35,Z 491.568,A -85,B 0,C 180,E1 -6041.068,E2 -6041.068} C_VEL
LIN {X 0,Y 504.166,Z 417.551,A -85,B 0,C 180,E1 -6042.196,E2 -6042.196} C_VEL
LIN {X 0,Y 505.47,Z 302.254,A -85,B 0,C 180,E1 -6043.916,E2 -6043.916} C_VEL
LIN {X 0,Y 503.81,Z 295.145,A -85,B 0,C 180,E1 -6044.122,E2 -6044.122} C_VEL
LIN {X 0,Y 499.116,Z 284.656,A -85,B 0,C 180,E1 -6044.575,E2 -6044.575} C_VEL
LIN {X 0,Y 495.763,Z 273.044,A -85,B 0,C 180,E1 -6046.15,E2 -6046.15} C_VEL
LIN {X 0,Y 495.771,Z 273.042,A -85,B 0,C 180,E1 -6049.029,E2 -6049.029} C_VEL
LIN {X 0,Y 495.743,Z 273.043,A -85,B 0,C 180,E1 -6051.629,E2 -6051.629} C_VEL
LIN {X 0,Y 495.716,Z 273.053,A -85,B 0,C 180,E1 -6054.277,E2 -6054.277} C_VEL
LIN {X 0,Y 495.721,Z 273.046,A -85,B 0,C 180,E1 -6056.98,E2 -6056.98} C_VEL
LIN {X 0,Y 495.747,Z 273.049,A -85,B 0,C 180,E1 -6060.142,E2 -6060.142} C_VEL
LIN {X 0,Y 495.73,Z 273.044,A -85,B 0,C 180,E1 -6063.232,E2 -6063.232} C_VEL
LIN {X 0,Y 495.676,Z 273.056,A -85,B 0,C 180,E1 -6066.081,E2 -6066.081} C_VEL
LIN {X 0,Y 495.723,Z 273.043,A -85,B 0,C 180,E1 -6068.761,E2 -6068.761} C_VEL
LIN {X 0,Y 495.701,Z 273.05,A -85,B 0,C 180,E1 -6071.787,E2 -6071.787} C_VEL
LIN {X 0,Y 495.733,Z 273.043,A -85,B 0,C 180,E1 -6075.141,E2 -6075.141} C_VEL
LIN {X 0,Y 495.702,Z 273.051,A -85,B 0,C 180,E1 -6078.213,E2 -6078.213} C_VEL
LIN {X 0,Y 495.721,Z 273.042,A -85,B 0,C 180,E1 -6081.405,E2 -6081.405} C_VEL
LIN {X 0,Y 495.729,Z 273.033,A -85,B 0,C 180,E1 -6084.46,E2 -6084.46} C_VEL
LIN {X 0,Y 495.752,Z 273.042,A -85,B 0,C 180,E1 -6087.404,E2 -6087.404} C_VEL
LIN {X 0,Y 495.757,Z 273.035,A -85,B 0,C 180,E1 -6090.252,E2 -6090.252} C_VEL
LIN {X 0,Y 495.739,Z 273.044,A -85,B 0,C 180,E1 -6093.27,E2 -6093.27} C_VEL
LIN {X 0,Y 495.741,Z 273.036,A -85,B 0,C 180,E1 -6096.612,E2 -6096.612} C_VEL
LIN {X 0,Y 495.781,Z 273.04,A -85,B 0,C 180,E1 -6099.324,E2 -6099.324} C_VEL
LIN {X 0,Y 495.781,Z 273.036,A -85,B 0,C 180,E1 -6101.828,E2 -6101.828} C_VEL
LIN {X 0,Y 495.825,Z 273.031,A -85,B 0,C 180,E1 -6104.548,E2 -6104.548} C_VEL
LIN {X 0,Y 495.83,Z 273.028,A -85,B 0,C 180,E1 -6107.965,E2 -6107.965} C_VEL
LIN {X 0,Y 495.832,Z 273.032,A -85,B 0,C 180,E1 -6111.03,E2 -6111.03} C_VEL
LIN {X 0,Y 495.865,Z 273.027,A -85,B 0,C 180,E1 -6113.489,E2 -6113.489} C_VEL
LIN {X 0,Y 495.72,Z 273.046,A -85,B 0,C 180,E1 -6115.935,E2 -6115.935} C_VEL
LIN {X 0,Y 495.987,Z 273.017,A -85,B 0,C 180,E1 -6117.563,E2 -6117.563} C_VEL
LIN {X 0,Y 495.999,Z 273.003,A -85,B 0,C 180,E1 -6120,E2 -6120} C_VEL
LIN {X 0,Y 495.993,Z 273.009,A -85,B 0,C 180,E1 -6122.436,E2 -6122.436} C_VEL
LIN {X 0,Y 495.885,Z 273.02,A -85,B 0,C 180,E1 -6125.693,E2 -6125.693} C_VEL
LIN {X 0,Y 495.842,Z 273.028,A -85,B 0,C 180,E1 -6128.969,E2 -6128.969} C_VEL
LIN {X 0,Y 495.829,Z 273.029,A -85,B 0,C 180,E1 -6132.034,E2 -6132.034} C_VEL
LIN {X 0,Y 495.824,Z 273.036,A -85,B 0,C 180,E1 -6135.451,E2 -6135.451} C_VEL
LIN {X 0,Y 495.778,Z 273.037,A -85,B 0,C 180,E1 -6138.237,E2 -6138.237} C_VEL
LIN {X 0,Y 495.774,Z 273.041,A -85,B 0,C 180,E1 -6140.756,E2 -6140.756} C_VEL
LIN {X 0,Y 495.751,Z 273.047,A -85,B 0,C 180,E1 -6143.387,E2 -6143.387} C_VEL
LIN {X 0,Y 495.79,Z 273.036,A -85,B 0,C 180,E1 -6146.067,E2 -6146.067} C_VEL
LIN {X 0,Y 495.771,Z 273.042,A -85,B 0,C 180,E1 -6148.814,E2 -6148.814} C_VEL
LIN {X 0,Y 495.754,Z 273.042,A -85,B 0,C 180,E1 -6151.725,E2 -6151.725} C_VEL
LIN {X 0,Y 495.773,Z 273.042,A -85,B 0,C 180,E1 -6154.695,E2 -6154.695} C_VEL
LIN {X 0,Y 495.73,Z 273.044,A -85,B 0,C 180,E1 -6157.561,E2 -6157.561} C_VEL
LIN {X 0,Y 495.766,Z 273.041,A -85,B 0,C 180,E1 -6160.7,E2 -6160.7} C_VEL
LIN {X 0,Y 495.733,Z 273.042,A -85,B 0,C 180,E1 -6163.695,E2 -6163.695} C_VEL
LIN {X 0,Y 495.734,Z 273.046,A -85,B 0,C 180,E1 -6166.304,E2 -6166.304} C_VEL
LIN {X 0,Y 495.766,Z 273.043,A -85,B 0,C 180,E1 -6169.3,E2 -6169.3} C_VEL
LIN {X 0,Y 495.728,Z 273.048,A -85,B 0,C 180,E1 -6172.438,E2 -6172.438} C_VEL
LIN {X 0,Y 495.776,Z 273.04,A -85,B 0,C 180,E1 -6175.457,E2 -6175.457} C_VEL
LIN {X 0,Y 495.759,Z 273.05,A -85,B 0,C 180,E1 -6178.428,E2 -6178.428} C_VEL
LIN {X 0,Y 502.107,Z 294.155,A -85,B 0,C 180,E1 -6181.011,E2 -6181.011} C_VEL
LIN {X 0,Y 502.401,Z 296.405,A -85,B 0,C 180,E1 -6181.258,E2 -6181.258} C_VEL
LIN {X 0,Y 501.734,Z 310.49,A -85,B 0,C 180,E1 -6182.63,E2 -6182.63} C_VEL
LIN {X 0,Y 505.338,Z 330.446,A -85,B 0,C 180,E1 -6183.145,E2 -6183.145} C_VEL
LIN {X 0,Y 503.268,Z 515.785,A -85,B 0,C 180,E1 -6185.919,E2 -6185.919} C_VEL
LIN {X 0,Y 502.795,Z 532.312,A -85,B 0,C 180,E1 -6186.305,E2 -6186.305} C_VEL
LIN {X 0,Y 502.191,Z 549.23,A -85,B 0,C 180,E1 -6186.876,E2 -6186.876} C_VEL
LIN {X 0,Y 501.466,Z 564.285,A -85,B 0,C 180,E1 -6187.536,E2 -6187.536} C_VEL
LIN {X 0,Y 500.674,Z 579.946,A -85,B 0,C 180,E1 -6188.404,E2 -6188.404} C_VEL
LIN {X 0,Y 499.887,Z 593.437,A -85,B 0,C 180,E1 -6189.315,E2 -6189.315} C_VEL
LIN {X 0,Y 498.974,Z 607.482,A -85,B 0,C 180,E1 -6190.434,E2 -6190.434} C_VEL
LIN {X 0,Y 498.136,Z 620.916,A -85,B 0,C 180,E1 -6191.705,E2 -6191.705} C_VEL
LIN {X 0,Y 497.402,Z 632.173,A -85,B 0,C 180,E1 -6192.951,E2 -6192.951} C_VEL
LIN {X 0,Y 496.716,Z 643.407,A -85,B 0,C 180,E1 -6194.405,E2 -6194.405} C_VEL
LIN {X 0,Y 496.209,Z 653.051,A -85,B 0,C 180,E1 -6195.859,E2 -6195.859} C_VEL
LIN {X 0,Y 495.823,Z 662.428,A -85,B 0,C 180,E1 -6197.517,E2 -6197.517} C_VEL
LIN {X 0,Y 495.452,Z 671.112,A -85,B 0,C 180,E1 -6199.374,E2 -6199.374} C_VEL
LIN {X 0,Y 495.164,Z 678.804,A -85,B 0,C 180,E1 -6201.429,E2 -6201.429} C_VEL
LIN {X 0,Y 495.111,Z 683.581,A -85,B 0,C 180,E1 -6203.07,E2 -6203.07} C_VEL
LIN {X 0,Y 495.034,Z 686.487,A -85,B 0,C 180,E1 -6204.297,E2 -6204.297} C_VEL
LIN {X 0,Y 494.984,Z 689.438,A -85,B 0,C 180,E1 -6205.929,E2 -6205.929} C_VEL
LIN {X 0,Y 494.967,Z 691.379,A -85,B 0,C 180,E1 -6207.559,E2 -6207.559} C_VEL
LIN {X 0,Y 494.906,Z 692.34,A -85,B 0,C 180,E1 -6209.186,E2 -6209.186} C_VEL
LIN {X 0,Y 494.906,Z 692.338,A -85,B 0,C 180,E1 -6210.814,E2 -6210.814} C_VEL
LIN {X 0,Y 494.967,Z 691.373,A -85,B 0,C 180,E1 -6212.441,E2 -6212.441} C_VEL
LIN {X 0,Y 494.984,Z 689.427,A -85,B 0,C 180,E1 -6214.071,E2 -6214.071} C_VEL
LIN {X 0,Y 495.034,Z 686.476,A -85,B 0,C 180,E1 -6215.704,E2 -6215.704} C_VEL
LIN {X 0,Y 495.145,Z 682.489,A -85,B 0,C 180,E1 -6217.339,E2 -6217.339} C_VEL
LIN {X 0,Y 495.206,Z 677.35,A -85,B 0,C 180,E1 -6218.981,E2 -6218.981} C_VEL
LIN {X 0,Y 495.452,Z 671.082,A -85,B 0,C 180,E1 -6220.627,E2 -6220.627} C_VEL
LIN {X 0,Y 495.818,Z 662.39,A -85,B 0,C 180,E1 -6222.484,E2 -6222.484} C_VEL
LIN {X 0,Y 496.208,Z 653.004,A -85,B 0,C 180,E1 -6224.142,E2 -6224.142} C_VEL
LIN {X 0,Y 496.749,Z 643.351,A -85,B 0,C 180,E1 -6225.594,E2 -6225.594} C_VEL
LIN {X 0,Y 497.402,Z 632.102,A -85,B 0,C 180,E1 -6227.049,E2 -6227.049} C_VEL
LIN {X 0,Y 498.184,Z 619.851,A -85,B 0,C 180,E1 -6228.4,E2 -6228.4} C_VEL
LIN {X 0,Y 498.995,Z 606.335,A -85,B 0,C 180,E1 -6229.661,E2 -6229.661} C_VEL
LIN {X 0,Y 499.906,Z 591.892,A -85,B 0,C 180,E1 -6230.792,E2 -6230.792} C_VEL
LIN {X 0,Y 500.783,Z 576.69,A -85,B 0,C 180,E1 -6231.782,E2 -6231.782} C_VEL
LIN {X 0,Y 501.585,Z 560.902,A -85,B 0,C 180,E1 -6232.62,E2 -6232.62} C_VEL
LIN {X 0,Y 502.373,Z 545.135,A -85,B 0,C 180,E1 -6233.279,E2 -6233.279} C_VEL
LIN {X 0,Y 502.924,Z 528.533,A -85,B 0,C 180,E1 -6233.798,E2 -6233.798} C_VEL
LIN {X 0,Y 503.339,Z 512.699,A -85,B 0,C 180,E1 -6234.133,E2 -6234.133} C_VEL
LIN {X 0,Y 505.358,Z 330.217,A -85,B 0,C 180,E1 -6236.871,E2 -6236.871} C_VEL
LIN {X 0,Y 501.716,Z 309.932,A -85,B 0,C 180,E1 -6237.418,E2 -6237.418} C_VEL
LIN {X 0,Y 502.489,Z 295.607,A -85,B 0,C 180,E1 -6238.851,E2 -6238.851} C_VEL
LIN {X 0,Y 498.308,Z 281.199,A -85,B 0,C 180,E1 -6240.647,E2 -6240.647} C_VEL
LIN {X 0,Y 495.754,Z 273.045,A -85,B 0,C 180,E1 -6241.726,E2 -6241.726} C_VEL
LIN {X 0,Y 495.768,Z 273.041,A -85,B 0,C 180,E1 -6244.694,E2 -6244.694} C_VEL
LIN {X 0,Y 495.729,Z 273.05,A -85,B 0,C 180,E1 -6247.562,E2 -6247.562} C_VEL
LIN {X 0,Y 495.766,Z 273.044,A -85,B 0,C 180,E1 -6250.7,E2 -6250.7} C_VEL
LIN {X 0,Y 495.735,Z 273.045,A -85,B 0,C 180,E1 -6253.696,E2 -6253.696} C_VEL
LIN {X 0,Y 495.729,Z 273.044,A -85,B 0,C 180,E1 -6256.306,E2 -6256.306} C_VEL
LIN {X 0,Y 495.767,Z 273.041,A -85,B 0,C 180,E1 -6259.301,E2 -6259.301} C_VEL
LIN {X 0,Y 495.73,Z 273.041,A -85,B 0,C 180,E1 -6262.439,E2 -6262.439} C_VEL
LIN {X 0,Y 495.778,Z 273.037,A -85,B 0,C 180,E1 -6265.457,E2 -6265.457} C_VEL
LIN {X 0,Y 495.755,Z 273.038,A -85,B 0,C 180,E1 -6268.364,E2 -6268.364} C_VEL
LIN {X 0,Y 495.788,Z 273.026,A -85,B 0,C 180,E1 -6271.507,E2 -6271.507} C_VEL
LIN {X 0,Y 495.792,Z 273.035,A -85,B 0,C 180,E1 -6273.933,E2 -6273.933} C_VEL
LIN {X 0,Y 495.762,Z 273.032,A -85,B 0,C 180,E1 -6277.139,E2 -6277.139} C_VEL
LIN {X 0,Y 495.772,Z 273.039,A -85,B 0,C 180,E1 -6280.11,E2 -6280.11} C_VEL
LIN {X 0,Y 495.781,Z 273.031,A -85,B 0,C 180,E1 -6282.682,E2 -6282.682} C_VEL
LIN {X 0,Y 495.79,Z 273.038,A -85,B 0,C 180,E1 -6285.218,E2 -6285.218} C_VEL
LIN {X 0,Y 495.853,Z 273.023,A -85,B 0,C 180,E1 -6288.555,E2 -6288.555} C_VEL
LIN {X 0,Y 495.832,Z 273.03,A -85,B 0,C 180,E1 -6291.852,E2 -6291.852} C_VEL
LIN {X 0,Y 495.833,Z 273.018,A -85,B 0,C 180,E1 -6295.122,E2 -6295.122} C_VEL
LIN {X 0,Y 495.989,Z 273.009,A -85,B 0,C 180,E1 -6297.564,E2 -6297.564} C_VEL
LIN {X 0,Y 495.944,Z 273.01,A -85,B 0,C 180,E1 -6300.812,E2 -6300.812} C_VEL
LIN {X 0,Y 495.981,Z 273.005,A -85,B 0,C 180,E1 -6302.437,E2 -6302.437} C_VEL
LIN {X 0,Y 495.872,Z 273.027,A -85,B 0,C 180,E1 -6305.694,E2 -6305.694} C_VEL
LIN {X 0,Y 495.816,Z 273.026,A -85,B 0,C 180,E1 -6308.149,E2 -6308.149} C_VEL
LIN {X 0,Y 495.853,Z 273.028,A -85,B 0,C 180,E1 -6311.446,E2 -6311.446} C_VEL
LIN {X 0,Y 495.782,Z 273.036,A -85,B 0,C 180,E1 -6314.784,E2 -6314.784} C_VEL
LIN {X 0,Y 495.775,Z 273.035,A -85,B 0,C 180,E1 -6318.235,E2 -6318.235} C_VEL
LIN {X 0,Y 495.777,Z 273.039,A -85,B 0,C 180,E1 -6320.757,E2 -6320.757} C_VEL
LIN {X 0,Y 495.736,Z 273.039,A -85,B 0,C 180,E1 -6323.388,E2 -6323.388} C_VEL
LIN {X 0,Y 495.709,Z 273.053,A -85,B 0,C 180,E1 -6326.073,E2 -6326.073} C_VEL
LIN {X 0,Y 495.698,Z 273.046,A -85,B 0,C 180,E1 -6328.82,E2 -6328.82} C_VEL
LIN {X 0,Y 495.732,Z 273.045,A -85,B 0,C 180,E1 -6331.72,E2 -6331.72} C_VEL
LIN {X 0,Y 495.739,Z 273.042,A -85,B 0,C 180,E1 -6334.688,E2 -6334.688} C_VEL
LIN {X 0,Y 495.692,Z 273.055,A -85,B 0,C 180,E1 -6337.566,E2 -6337.566} C_VEL
LIN {X 0,Y 495.71,Z 273.053,A -85,B 0,C 180,E1 -6340.04,E2 -6340.04} C_VEL
LIN {X 0,Y 495.692,Z 273.05,A -85,B 0,C 180,E1 -6342.887,E2 -6342.887} C_VEL
LIN {X 0,Y 495.716,Z 273.049,A -85,B 0,C 180,E1 -6345.997,E2 -6345.997} C_VEL
LIN {X 0,Y 495.717,Z 273.148,A -85,B 0,C 180,E1 -6347.821,E2 -6347.821} C_VEL
LIN {X 0,Y 499.217,Z 285.004,A -85,B 0,C 180,E1 -6349.484,E2 -6349.484} C_VEL
LIN {X 0,Y 504.382,Z 296.396,A -85,B 0,C 180,E1 -6349.99,E2 -6349.99} C_VEL
LIN {X 0,Y 505.56,Z 303.01,A -85,B 0,C 180,E1 -6350.166,E2 -6350.166} C_VEL
LIN {X 0,Y 505.018,Z 351.105,A -85,B 0,C 180,E1 -6350.892,E2 -6350.892} C_VEL
LIN {X 0,Y 504.478,Z 356.953,A -85,B 0,C 180,E1 -6350.953,E2 -6350.953} C_VEL
LIN {X 0,Y 501.792,Z 366.498,A -85,B 0,C 180,E1 -6350.947,E2 -6350.947} C_VEL
LIN {X 0,Y 498.993,Z 376.049,A -85,B 0,C 180,E1 -6350.935,E2 -6350.935} C_VEL
LIN {X 0,Y 498.284,Z 381.912,A -85,B 0,C 180,E1 -6350.987,E2 -6350.987} C_VEL
LIN {X 0,Y 496.927,Z 491.51,A -85,B 0,C 180,E1 -6352.672,E2 -6352.672} C_VEL
LIN {X 0,Y 496.406,Z 508.904,A -85,B 0,C 180,E1 -6353.119,E2 -6353.119} C_VEL
LIN {X 0,Y 495.762,Z 525.015,A -85,B 0,C 180,E1 -6353.707,E2 -6353.707} C_VEL
LIN {X 0,Y 494.959,Z 540.893,A -85,B 0,C 180,E1 -6354.459,E2 -6354.459} C_VEL
LIN {X 0,Y 494.139,Z 555.581,A -85,B 0,C 180,E1 -6355.326,E2 -6355.326} C_VEL
LIN {X 0,Y 493.221,Z 570.119,A -85,B 0,C 180,E1 -6356.362,E2 -6356.362} C_VEL
LIN {X 0,Y 492.242,Z 584.311,A -85,B 0,C 180,E1 -6357.581,E2 -6357.581} C_VEL
LIN {X 0,Y 491.325,Z 597.065,A -85,B 0,C 180,E1 -6358.886,E2 -6358.886} C_VEL
LIN {X 0,Y 490.47,Z 609.397,A -85,B 0,C 180,E1 -6360.373,E2 -6360.373} C_VEL
LIN {X 0,Y 489.738,Z 620.57,A -85,B 0,C 180,E1 -6361.967,E2 -6361.967} C_VEL
LIN {X 0,Y 489.159,Z 629.998,A -85,B 0,C 180,E1 -6363.551,E2 -6363.551} C_VEL
LIN {X 0,Y 488.66,Z 638.96,A -85,B 0,C 180,E1 -6365.349,E2 -6365.349} C_VEL
LIN {X 0,Y 488.33,Z 646.225,A -85,B 0,C 180,E1 -6367.134,E2 -6367.134} C_VEL
LIN {X 0,Y 488.13,Z 652.061,A -85,B 0,C 180,E1 -6368.903,E2 -6368.903} C_VEL
LIN {X 0,Y 487.973,Z 656.649,A -85,B 0,C 180,E1 -6370.655,E2 -6370.655} C_VEL
LIN {X 0,Y 487.839,Z 660.015,A -85,B 0,C 180,E1 -6372.39,E2 -6372.39} C_VEL
LIN {X 0,Y 487.77,Z 662.278,A -85,B 0,C 180,E1 -6374.112,E2 -6374.112} C_VEL
LIN {X 0,Y 487.82,Z 663.531,A -85,B 0,C 180,E1 -6375.823,E2 -6375.823} C_VEL
LIN {X 0,Y 487.836,Z 663.715,A -85,B 0,C 180,E1 -6377.52,E2 -6377.52} C_VEL
LIN {X 0,Y 487.855,Z 662.987,A -85,B 0,C 180,E1 -6379.206,E2 -6379.206} C_VEL
LIN {X 0,Y 487.833,Z 661.199,A -85,B 0,C 180,E1 -6380.882,E2 -6380.882} C_VEL
LIN {X 0,Y 487.914,Z 658.51,A -85,B 0,C 180,E1 -6382.551,E2 -6382.551} C_VEL
LIN {X 0,Y 488.088,Z 654.709,A -85,B 0,C 180,E1 -6384.215,E2 -6384.215} C_VEL
LIN {X 0,Y 488.187,Z 649.942,A -85,B 0,C 180,E1 -6385.872,E2 -6385.872} C_VEL
LIN {X 0,Y 488.351,Z 644.019,A -85,B 0,C 180,E1 -6387.525,E2 -6387.525} C_VEL
LIN {X 0,Y 488.752,Z 636.855,A -85,B 0,C 180,E1 -6389.176,E2 -6389.176} C_VEL
LIN {X 0,Y 489.167,Z 628.385,A -85,B 0,C 180,E1 -6390.823,E2 -6390.823} C_VEL
LIN {X 0,Y 489.826,Z 618.32,A -85,B 0,C 180,E1 -6392.467,E2 -6392.467} C_VEL
LIN {X 0,Y 490.714,Z 606.325,A -85,B 0,C 180,E1 -6394.106,E2 -6394.106} C_VEL
LIN {X 0,Y 491.566,Z 593.897,A -85,B 0,C 180,E1 -6395.538,E2 -6395.538} C_VEL
LIN {X 0,Y 492.322,Z 582.541,A -85,B 0,C 180,E1 -6396.66,E2 -6396.66} C_VEL
LIN {X 0,Y 493.199,Z 569.357,A -85,B 0,C 180,E1 -6397.78,E2 -6397.78} C_VEL
LIN {X 0,Y 494.092,Z 554.987,A -85,B 0,C 180,E1 -6398.795,E2 -6398.795} C_VEL
LIN {X 0,Y 494.844,Z 541.181,A -85,B 0,C 180,E1 -6399.606,E2 -6399.606} C_VEL
LIN {X 0,Y 495.622,Z 525.235,A -85,B 0,C 180,E1 -6400.364,E2 -6400.364} C_VEL
LIN {X 0,Y 496.311,Z 509.389,A -85,B 0,C 180,E1 -6400.943,E2 -6400.943} C_VEL
LIN {X 0,Y 496.847,Z 492.868,A -85,B 0,C 180,E1 -6401.37,E2 -6401.37} C_VEL
LIN {X 0,Y 497.293,Z 461.398,A -85,B 0,C 180,E1 -6401.877,E2 -6401.877} C_VEL
LIN {X 0,Y 499.101,Z 304.083,A -85,B 0,C 180,E1 -6404.251,E2 -6404.251} C_VEL
LIN {X 0,Y 497.906,Z 298.214,A -85,B 0,C 180,E1 -6404.413,E2 -6404.413} C_VEL
LIN {X 0,Y 491.929,Z 284.906,A -85,B 0,C 180,E1 -6404.99,E2 -6404.99} C_VEL
LIN {X 0,Y 488.716,Z 273.924,A -85,B 0,C 180,E1 -6406.508,E2 -6406.508} C_VEL
LIN {X 0,Y 488.734,Z 273.918,A -85,B 0,C 180,E1 -6409.314,E2 -6409.314} C_VEL
LIN {X 0,Y 488.7,Z 273.918,A -85,B 0,C 180,E1 -6411.957,E2 -6411.957} C_VEL
LIN {X 0,Y 488.699,Z 273.919,A -85,B 0,C 180,E1 -6415.04,E2 -6415.04} C_VEL
LIN {X 0,Y 488.694,Z 273.927,A -85,B 0,C 180,E1 -6418.332,E2 -6418.332} C_VEL
LIN {X 0,Y 488.68,Z 273.924,A -85,B 0,C 180,E1 -6421.181,E2 -6421.181} C_VEL
LIN {X 0,Y 488.704,Z 273.923,A -85,B 0,C 180,E1 -6424.115,E2 -6424.115} C_VEL
LIN {X 0,Y 488.636,Z 273.927,A -85,B 0,C 180,E1 -6427.163,E2 -6427.163} C_VEL
LIN {X 0,Y 488.665,Z 273.927,A -85,B 0,C 180,E1 -6430.336,E2 -6430.336} C_VEL
LIN {X 0,Y 488.666,Z 273.926,A -85,B 0,C 180,E1 -6433.657,E2 -6433.657} C_VEL
LIN {X 0,Y 488.666,Z 273.922,A -85,B 0,C 180,E1 -6436.343,E2 -6436.343} C_VEL
LIN {X 0,Y 488.669,Z 273.928,A -85,B 0,C 180,E1 -6439.669,E2 -6439.669} C_VEL
LIN {X 0,Y 488.648,Z 273.91,A -85,B 0,C 180,E1 -6442.283,E2 -6442.283} C_VEL
LIN {X 0,Y 488.714,Z 273.905,A -85,B 0,C 180,E1 -6445.054,E2 -6445.054} C_VEL
LIN {X 0,Y 488.699,Z 273.924,A -85,B 0,C 180,E1 -6448.047,E2 -6448.047} C_VEL
LIN {X 0,Y 488.7,Z 273.912,A -85,B 0,C 180,E1 -6450.728,E2 -6450.728} C_VEL
LIN {X 0,Y 488.683,Z 273.926,A -85,B 0,C 180,E1 -6453.523,E2 -6453.523} C_VEL
LIN {X 0,Y 488.671,Z 273.918,A -85,B 0,C 180,E1 -6456.253,E2 -6456.253} C_VEL
LIN {X 0,Y 488.749,Z 273.915,A -85,B 0,C 180,E1 -6459.175,E2 -6459.175} C_VEL
LIN {X 0,Y 488.749,Z 273.913,A -85,B 0,C 180,E1 -6461.632,E2 -6461.632} C_VEL
LIN {X 0,Y 488.758,Z 273.913,A -85,B 0,C 180,E1 -6464.999,E2 -6464.999} C_VEL
LIN {X 0,Y 488.807,Z 273.899,A -85,B 0,C 180,E1 -6468.387,E2 -6468.387} C_VEL
LIN {X 0,Y 488.785,Z 273.912,A -85,B 0,C 180,E1 -6471.733,E2 -6471.733} C_VEL
LIN {X 0,Y 488.849,Z 273.893,A -85,B 0,C 180,E1 -6474.224,E2 -6474.224} C_VEL
LIN {X 0,Y 488.953,Z 273.894,A -85,B 0,C 180,E1 -6477.528,E2 -6477.528} C_VEL
LIN {X 0,Y 488.97,Z 273.878,A -85,B 0,C 180,E1 -6480,E2 -6480} C_VEL
LIN {X 0,Y 488.961,Z 273.885,A -85,B 0,C 180,E1 -6482.471,E2 -6482.471} C_VEL
LIN {X 0,Y 488.842,Z 273.896,A -85,B 0,C 180,E1 -6485.775,E2 -6485.775} C_VEL
LIN {X 0,Y 488.818,Z 273.899,A -85,B 0,C 180,E1 -6488.266,E2 -6488.266} C_VEL
LIN {X 0,Y 488.806,Z 273.907,A -85,B 0,C 180,E1 -6491.612,E2 -6491.612} C_VEL
LIN {X 0,Y 488.761,Z 273.917,A -85,B 0,C 180,E1 -6495,E2 -6495} C_VEL
LIN {X 0,Y 488.747,Z 273.914,A -85,B 0,C 180,E1 -6498.442,E2 -6498.442} C_VEL
LIN {X 0,Y 488.707,Z 273.926,A -85,B 0,C 180,E1 -6501.07,E2 -6501.07} C_VEL
LIN {X 0,Y 488.693,Z 273.922,A -85,B 0,C 180,E1 -6503.745,E2 -6503.745} C_VEL
LIN {X 0,Y 488.791,Z 273.915,A -85,B 0,C 180,E1 -6506.943,E2 -6506.943} C_VEL
LIN {X 0,Y 488.709,Z 273.919,A -85,B 0,C 180,E1 -6510.362,E2 -6510.362} C_VEL
LIN {X 0,Y 488.734,Z 273.917,A -85,B 0,C 180,E1 -6513.484,E2 -6513.484} C_VEL
LIN {X 0,Y 488.686,Z 273.919,A -85,B 0,C 180,E1 -6516.355,E2 -6516.355} C_VEL
LIN {X 0,Y 488.701,Z 273.922,A -85,B 0,C 180,E1 -6519.254,E2 -6519.254} C_VEL
LIN {X 0,Y 488.722,Z 273.918,A -85,B 0,C 180,E1 -6521.602,E2 -6521.602} C_VEL
LIN {X 0,Y 488.711,Z 273.921,A -85,B 0,C 180,E1 -6524.801,E2 -6524.801} C_VEL
LIN {X 0,Y 488.694,Z 273.92,A -85,B 0,C 180,E1 -6527.475,E2 -6527.475} C_VEL
LIN {X 0,Y 488.731,Z 273.917,A -85,B 0,C 180,E1 -6529.676,E2 -6529.676} C_VEL
LIN {X 0,Y 488.678,Z 273.927,A -85,B 0,C 180,E1 -6532.841,E2 -6532.841} C_VEL
LIN {X 0,Y 488.728,Z 273.917,A -85,B 0,C 180,E1 -6535.887,E2 -6535.887} C_VEL
LIN {X 0,Y 488.732,Z 273.946,A -85,B 0,C 180,E1 -6538.067,E2 -6538.067} C_VEL
LIN {X 0,Y 495.218,Z 295.546,A -85,B 0,C 180,E1 -6540.752,E2 -6540.752} C_VEL
LIN {X 0,Y 495.763,Z 297.496,A -85,B 0,C 180,E1 -6540.986,E2 -6540.986} C_VEL
LIN {X 0,Y 495.116,Z 310.2,A -85,B 0,C 180,E1 -6542.244,E2 -6542.244} C_VEL
LIN {X 0,Y 498.944,Z 332.168,A -85,B 0,C 180,E1 -6542.813,E2 -6542.813} C_VEL
LIN {X 0,Y 496.785,Z 515.416,A -85,B 0,C 180,E1 -6545.586,E2 -6545.586} C_VEL
LIN {X 0,Y 496.296,Z 531.971,A -85,B 0,C 180,E1 -6545.976,E2 -6545.976} C_VEL
LIN {X 0,Y 495.717,Z 547.637,A -85,B 0,C 180,E1 -6546.501,E2 -6546.501} C_VEL
LIN {X 0,Y 494.92,Z 563.242,A -85,B 0,C 180,E1 -6547.18,E2 -6547.18} C_VEL
LIN {X 0,Y 494.091,Z 578.503,A -85,B 0,C 180,E1 -6548.027,E2 -6548.027} C_VEL
LIN {X 0,Y 493.215,Z 591.775,A -85,B 0,C 180,E1 -6548.912,E2 -6548.912} C_VEL
LIN {X 0,Y 492.282,Z 606.328,A -85,B 0,C 180,E1 -6550.071,E2 -6550.071} C_VEL
LIN {X 0,Y 491.341,Z 619.713,A -85,B 0,C 180,E1 -6551.334,E2 -6551.334} C_VEL
LIN {X 0,Y 490.494,Z 631.954,A -85,B 0,C 180,E1 -6552.704,E2 -6552.704} C_VEL
LIN {X 0,Y 489.754,Z 643.19,A -85,B 0,C 180,E1 -6554.178,E2 -6554.178} C_VEL
LIN {X 0,Y 489.216,Z 652.838,A -85,B 0,C 180,E1 -6555.652,E2 -6555.652} C_VEL
LIN {X 0,Y 488.788,Z 662.216,A -85,B 0,C 180,E1 -6557.334,E2 -6557.334} C_VEL
LIN {X 0,Y 488.391,Z 670.901,A -85,B 0,C 180,E1 -6559.218,E2 -6559.218} C_VEL
LIN {X 0,Y 488.09,Z 678.595,A -85,B 0,C 180,E1 -6561.304,E2 -6561.304} C_VEL
LIN {X 0,Y 487.994,Z 684.449,A -85,B 0,C 180,E1 -6563.384,E2 -6563.384} C_VEL
LIN {X 0,Y 487.907,Z 687.872,A -85,B 0,C 180,E1 -6565.042,E2 -6565.042} C_VEL
LIN {X 0,Y 487.944,Z 690.36,A -85,B 0,C 180,E1 -6566.697,E2 -6566.697} C_VEL
LIN {X 0,Y 487.883,Z 691.762,A -85,B 0,C 180,E1 -6568.349,E2 -6568.349} C_VEL
LIN {X 0,Y 487.814,Z 692.286,A -85,B 0,C 180,E1 -6570,E2 -6570} C_VEL
LIN {X 0,Y 487.883,Z 691.756,A -85,B 0,C 180,E1 -6571.651,E2 -6571.651} C_VEL
LIN {X 0,Y 487.944,Z 690.349,A -85,B 0,C 180,E1 -6573.303,E2 -6573.303} C_VEL
LIN {X 0,Y 487.907,Z 687.856,A -85,B 0,C 180,E1 -6574.958,E2 -6574.958} C_VEL
LIN {X 0,Y 487.994,Z 684.432,A -85,B 0,C 180,E1 -6576.616,E2 -6576.616} C_VEL
LIN {X 0,Y 488.09,Z 678.569,A -85,B 0,C 180,E1 -6578.696,E2 -6578.696} C_VEL
LIN {X 0,Y 488.391,Z 670.863,A -85,B 0,C 180,E1 -6580.782,E2 -6580.782} C_VEL
LIN {X 0,Y 488.736,Z 663.188,A -85,B 0,C 180,E1 -6582.457,E2 -6582.457} C_VEL
LIN {X 0,Y 489.16,Z 654.023,A -85,B 0,C 180,E1 -6584.137,E2 -6584.137} C_VEL
LIN {X 0,Y 489.732,Z 644.621,A -85,B 0,C 180,E1 -6585.609,E2 -6585.609} C_VEL
LIN {X 0,Y 490.378,Z 633.614,A -85,B 0,C 180,E1 -6587.086,E2 -6587.086} C_VEL
LIN {X 0,Y 491.171,Z 622.566,A -85,B 0,C 180,E1 -6588.348,E2 -6588.348} C_VEL
LIN {X 0,Y 491.896,Z 611.679,A -85,B 0,C 180,E1 -6589.443,E2 -6589.443} C_VEL
LIN {X 0,Y 492.875,Z 597.321,A -85,B 0,C 180,E1 -6590.666,E2 -6590.666} C_VEL
LIN {X 0,Y 493.652,Z 584.062,A -85,B 0,C 180,E1 -6591.616,E2 -6591.616} C_VEL
LIN {X 0,Y 494.637,Z 568.172,A -85,B 0,C 180,E1 -6592.559,E2 -6592.559} C_VEL
LIN {X 0,Y 495.445,Z 552.859,A -85,B 0,C 180,E1 -6593.292,E2 -6593.292} C_VEL
LIN {X 0,Y 496.175,Z 536.622,A -85,B 0,C 180,E1 -6593.892,E2 -6593.892} C_VEL
LIN {X 0,Y 496.681,Z 520.815,A -85,B 0,C 180,E1 -6594.31,E2 -6594.31} C_VEL
LIN {X 0,Y 497.147,Z 497.498,A -85,B 0,C 180,E1 -6594.703,E2 -6594.703} C_VEL
LIN {X 0,Y 499.065,Z 331.201,A -85,B 0,C 180,E1 -6597.231,E2 -6597.231} C_VEL
LIN {X 0,Y 495.217,Z 309.678,A -85,B 0,C 180,E1 -6597.83,E2 -6597.83} C_VEL
LIN {X 0,Y 495.893,Z 298.054,A -85,B 0,C 180,E1 -6599.011,E2 -6599.011} C_VEL
LIN {X 0,Y 492.472,Z 285.78,A -85,B 0,C 180,E1 -6600.555,E2 -6600.555} C_VEL
LIN {X 0,Y 488.702,Z 273.924,A -85,B 0,C 180,E1 -6602.147,E2 -6602.147} C_VEL
LIN {X 0,Y 488.716,Z 273.92,A -85,B 0,C 180,E1 -6605.115,E2 -6605.115} C_VEL
LIN {X 0,Y 488.68,Z 273.925,A -85,B 0,C 180,E1 -6608.2,E2 -6608.2} C_VEL
LIN {X 0,Y 488.718,Z 273.916,A -85,B 0,C 180,E1 -6611.415,E2 -6611.415} C_VEL
LIN {X 0,Y 488.702,Z 273.92,A -85,B 0,C 180,E1 -6614.025,E2 -6614.025} C_VEL
LIN {X 0,Y 488.709,Z 273.922,A -85,B 0,C 180,E1 -6617.174,E2 -6617.174} C_VEL
LIN {X 0,Y 488.733,Z 273.917,A -85,B 0,C 180,E1 -6619.677,E2 -6619.677} C_VEL
LIN {X 0,Y 488.679,Z 273.919,A -85,B 0,C 180,E1 -6622.842,E2 -6622.842} C_VEL
LIN {X 0,Y 488.73,Z 273.913,A -85,B 0,C 180,E1 -6625.888,E2 -6625.888} C_VEL
LIN {X 0,Y 488.693,Z 273.924,A -85,B 0,C 180,E1 -6628.821,E2 -6628.821} C_VEL
LIN {X 0,Y 488.745,Z 273.902,A -85,B 0,C 180,E1 -6631.672,E2 -6631.672} C_VEL
LIN {X 0,Y 488.749,Z 273.916,A -85,B 0,C 180,E1 -6634.445,E2 -6634.445} C_VEL
LIN {X 0,Y 488.725,Z 273.907,A -85,B 0,C 180,E1 -6637.154,E2 -6637.154} C_VEL
LIN {X 0,Y 488.726,Z 273.916,A -85,B 0,C 180,E1 -6639.811,E2 -6639.811} C_VEL
LIN {X 0,Y 488.729,Z 273.912,A -85,B 0,C 180,E1 -6642.424,E2 -6642.424} C_VEL
LIN {X 0,Y 488.762,Z 273.915,A -85,B 0,C 180,E1 -6645,E2 -6645} C_VEL
LIN {X 0,Y 488.807,Z 273.902,A -85,B 0,C 180,E1 -6648.388,E2 -6648.388} C_VEL
LIN {X 0,Y 488.782,Z 273.908,A -85,B 0,C 180,E1 -6651.733,E2 -6651.733} C_VEL
LIN {X 0,Y 488.832,Z 273.904,A -85,B 0,C 180,E1 -6654.224,E2 -6654.224} C_VEL
LIN {X 0,Y 488.956,Z 273.885,A -85,B 0,C 180,E1 -6657.529,E2 -6657.529} C_VEL
LIN {X 0,Y 488.97,Z 273.888,A -85,B 0,C 180,E1 -6660,E2 -6660} C_VEL
LIN {X 0,Y 488.947,Z 273.881,A -85,B 0,C 180,E1 -6662.472,E2 -6662.472} C_VEL
LIN {X 0,Y 488.829,Z 273.905,A -85,B 0,C 180,E1 -6665.777,E2 -6665.777} C_VEL
LIN {X 0,Y 488.764,Z 273.904,A -85,B 0,C 180,E1 -6668.268,E2 -6668.268} C_VEL
LIN {X 0,Y 488.808,Z 273.907,A -85,B 0,C 180,E1 -6671.613,E2 -6671.613} C_VEL
LIN {X 0,Y 488.752,Z 273.911,A -85,B 0,C 180,E1 -6675.001,E2 -6675.001} C_VEL
LIN {X 0,Y 488.747,Z 273.907,A -85,B 0,C 180,E1 -6678.443,E2 -6678.443} C_VEL
LIN {X 0,Y 488.709,Z 273.919,A -85,B 0,C 180,E1 -6681.071,E2 -6681.071} C_VEL
LIN {X 0,Y 488.665,Z 273.92,A -85,B 0,C 180,E1 -6683.747,E2 -6683.747} C_VEL
LIN {X 0,Y 488.67,Z 273.925,A -85,B 0,C 180,E1 -6686.478,E2 -6686.478} C_VEL
LIN {X 0,Y 488.662,Z 273.922,A -85,B 0,C 180,E1 -6689.275,E2 -6689.275} C_VEL
LIN {X 0,Y 488.681,Z 273.921,A -85,B 0,C 180,E1 -6692.149,E2 -6692.149} C_VEL
LIN {X 0,Y 488.696,Z 273.919,A -85,B 0,C 180,E1 -6695.117,E2 -6695.117} C_VEL
LIN {X 0,Y 488.647,Z 273.927,A -85,B 0,C 180,E1 -6698.204,E2 -6698.204} C_VEL
LIN {X 0,Y 488.645,Z 273.926,A -85,B 0,C 180,E1 -6701.423,E2 -6701.423} C_VEL
LIN {X 0,Y 488.699,Z 273.922,A -85,B 0,C 180,E1 -6704.804,E2 -6704.804} C_VEL
LIN {X 0,Y 488.666,Z 273.99,A -85,B 0,C 180,E1 -6707.402,E2 -6707.402} C_VEL
LIN {X 0,Y 492.139,Z 285.44,A -85,B 0,C 180,E1 -6709.036,E2 -6709.036} C_VEL
LIN {X 0,Y 498.441,Z 299.108,A -85,B 0,C 180,E1 -6709.666,E2 -6709.666} C_VEL
LIN {X 0,Y 499.306,Z 304.263,A -85,B 0,C 180,E1 -6709.804,E2 -6709.804} C_VEL
LIN {X 0,Y 498.284,Z 381.912,A -85,B 0,C 180,E1 -6710.987,E2 -6710.987} C_VEL
LIN {X 0,Y 497.604,Z 387.765,A -85,B 0,C 180,E1 -6711.04,E2 -6711.04} C_VEL
LIN {X 0,Y 492.233,Z 406.862,A -85,B 0,C 180,E1 -6711.028,E2 -6711.028} C_VEL
LIN {X 0,Y 491.596,Z 412.712,A -85,B 0,C 180,E1 -6711.084,E2 -6711.084} C_VEL
LIN {X 0,Y 490.525,Z 491.984,A -85,B 0,C 180,E1 -6712.327,E2 -6712.327} C_VEL
LIN {X 0,Y 489.958,Z 509.255,A -85,B 0,C 180,E1 -6712.777,E2 -6712.777} C_VEL
LIN {X 0,Y 489.32,Z 524.393,A -85,B 0,C 180,E1 -6713.335,E2 -6713.335} C_VEL
LIN {X 0,Y 488.475,Z 540.597,A -85,B 0,C 180,E1 -6714.105,E2 -6714.105} C_VEL
LIN {X 0,Y 487.597,Z 555.099,A -85,B 0,C 180,E1 -6714.963,E2 -6714.963} C_VEL
LIN {X 0,Y 486.633,Z 569.168,A -85,B 0,C 180,E1 -6715.97,E2 -6715.97} C_VEL
LIN {X 0,Y 485.713,Z 581.924,A -85,B 0,C 180,E1 -6717.06,E2 -6717.06} C_VEL
LIN {X 0,Y 484.692,Z 595.375,A -85,B 0,C 180,E1 -6718.412,E2 -6718.412} C_VEL
LIN {X 0,Y 483.874,Z 606.258,A -85,B 0,C 180,E1 -6719.687,E2 -6719.687} C_VEL
LIN {X 0,Y 483.033,Z 617.967,A -85,B 0,C 180,E1 -6721.305,E2 -6721.305} C_VEL
LIN {X 0,Y 482.35,Z 627.832,A -85,B 0,C 180,E1 -6722.925,E2 -6722.925} C_VEL
LIN {X 0,Y 481.883,Z 635.768,A -85,B 0,C 180,E1 -6724.451,E2 -6724.451} C_VEL
LIN {X 0,Y 481.516,Z 642.127,A -85,B 0,C 180,E1 -6725.878,E2 -6725.878} C_VEL
LIN {X 0,Y 481.182,Z 648.834,A -85,B 0,C 180,E1 -6727.682,E2 -6727.682} C_VEL
LIN {X 0,Y 481.023,Z 654.207,A -85,B 0,C 180,E1 -6729.473,E2 -6729.473} C_VEL
LIN {X 0,Y 480.838,Z 658.29,A -85,B 0,C 180,E1 -6731.243,E2 -6731.243} C_VEL
LIN {X 0,Y 480.702,Z 661.217,A -85,B 0,C 180,E1 -6732.998,E2 -6732.998} C_VEL
LIN {X 0,Y 480.705,Z 663.154,A -85,B 0,C 180,E1 -6734.784,E2 -6734.784} C_VEL
LIN {X 0,Y 480.702,Z 663.908,A -85,B 0,C 180,E1 -6736.472,E2 -6736.472} C_VEL
LIN {X 0,Y 480.844,Z 663.712,A -85,B 0,C 180,E1 -6738.316,E2 -6738.316} C_VEL
LIN {X 0,Y 480.732,Z 662.591,A -85,B 0,C 180,E1 -6739.896,E2 -6739.896} C_VEL
LIN {X 0,Y 480.78,Z 660.502,A -85,B 0,C 180,E1 -6741.594,E2 -6741.594} C_VEL
LIN {X 0,Y 480.956,Z 656.789,A -85,B 0,C 180,E1 -6743.546,E2 -6743.546} C_VEL
LIN {X 0,Y 481.056,Z 651.989,A -85,B 0,C 180,E1 -6745.391,E2 -6745.391} C_VEL
LIN {X 0,Y 481.263,Z 646.513,A -85,B 0,C 180,E1 -6747.07,E2 -6747.07} C_VEL
LIN {X 0,Y 481.606,Z 639.825,A -85,B 0,C 180,E1 -6748.746,E2 -6748.746} C_VEL
LIN {X 0,Y 482.016,Z 631.817,A -85,B 0,C 180,E1 -6750.418,E2 -6750.418} C_VEL
LIN {X 0,Y 482.647,Z 622.343,A -85,B 0,C 180,E1 -6752.086,E2 -6752.086} C_VEL
LIN {X 0,Y 483.404,Z 612.644,A -85,B 0,C 180,E1 -6753.542,E2 -6753.542} C_VEL
LIN {X 0,Y 484.234,Z 601.257,A -85,B 0,C 180,E1 -6754.996,E2 -6754.996} C_VEL
LIN {X 0,Y 485.11,Z 588.919,A -85,B 0,C 180,E1 -6756.342,E2 -6756.342} C_VEL
LIN {X 0,Y 486.063,Z 575.534,A -85,B 0,C 180,E1 -6757.582,E2 -6757.582} C_VEL
LIN {X 0,Y 487.052,Z 560.924,A -85,B 0,C 180,E1 -6758.714,E2 -6758.714} C_VEL
LIN {X 0,Y 488.013,Z 546.443,A -85,B 0,C 180,E1 -6759.637,E2 -6759.637} C_VEL
LIN {X 0,Y 488.815,Z 531.666,A -85,B 0,C 180,E1 -6760.406,E2 -6760.406} C_VEL
LIN {X 0,Y 489.52,Z 516.184,A -85,B 0,C 180,E1 -6761.045,E2 -6761.045} C_VEL
LIN {X 0,Y 490.136,Z 499.545,A -85,B 0,C 180,E1 -6761.554,E2 -6761.554} C_VEL
LIN {X 0,Y 490.539,Z 483.277,A -85,B 0,C 180,E1 -6761.885,E2 -6761.885} C_VEL
LIN {X 0,Y 492.733,Z 305.061,A -85,B 0,C 180,E1 -6764.605,E2 -6764.605} C_VEL
LIN {X 0,Y 491.864,Z 300.933,A -85,B 0,C 180,E1 -6764.722,E2 -6764.722} C_VEL
LIN {X 0,Y 484.716,Z 285.143,A -85,B 0,C 180,E1 -6765.417,E2 -6765.417} C_VEL
LIN {X 0,Y 481.65,Z 274.801,A -85,B 0,C 180,E1 -6766.885,E2 -6766.885} C_VEL
LIN {X 0,Y 481.7,Z 274.796,A -85,B 0,C 180,E1 -6769.607,E2 -6769.607} C_VEL
LIN {X 0,Y 481.651,Z 274.796,A -85,B 0,C 180,E1 -6772.295,E2 -6772.295} C_VEL
LIN {X 0,Y 481.662,Z 274.796,A -85,B 0,C 180,E1 -6775.222,E2 -6775.222} C_VEL
LIN {X 0,Y 481.648,Z 274.803,A -85,B 0,C 180,E1 -6777.835,E2 -6777.835} C_VEL
LIN {X 0,Y 481.631,Z 274.803,A -85,B 0,C 180,E1 -6780.712,E2 -6780.712} C_VEL
LIN {X 0,Y 481.652,Z 274.802,A -85,B 0,C 180,E1 -6783.724,E2 -6783.724} C_VEL
LIN {X 0,Y 481.599,Z 274.805,A -85,B 0,C 180,E1 -6786.749,E2 -6786.749} C_VEL
LIN {X 0,Y 481.629,Z 274.806,A -85,B 0,C 180,E1 -6789.945,E2 -6789.945} C_VEL
LIN {X 0,Y 481.616,Z 274.8,A -85,B 0,C 180,E1 -6793.302,E2 -6793.302} C_VEL
LIN {X 0,Y 481.65,Z 274.801,A -85,B 0,C 180,E1 -6795.642,E2 -6795.642} C_VEL
LIN {X 0,Y 481.605,Z 274.803,A -85,B 0,C 180,E1 -6798.952,E2 -6798.952} C_VEL
LIN {X 0,Y 481.63,Z 274.787,A -85,B 0,C 180,E1 -6801.997,E2 -6801.997} C_VEL
LIN {X 0,Y 481.679,Z 274.783,A -85,B 0,C 180,E1 -6805.316,E2 -6805.316} C_VEL
LIN {X 0,Y 481.64,Z 274.8,A -85,B 0,C 180,E1 -6808.311,E2 -6808.311} C_VEL
LIN {X 0,Y 481.659,Z 274.791,A -85,B 0,C 180,E1 -6811.215,E2 -6811.215} C_VEL
LIN {X 0,Y 481.63,Z 274.802,A -85,B 0,C 180,E1 -6814.038,E2 -6814.038} C_VEL
LIN {X 0,Y 481.676,Z 274.788,A -85,B 0,C 180,E1 -6816.812,E2 -6816.812} C_VEL
LIN {X 0,Y 481.697,Z 274.797,A -85,B 0,C 180,E1 -6819.502,E2 -6819.502} C_VEL
LIN {X 0,Y 481.689,Z 274.788,A -85,B 0,C 180,E1 -6822.157,E2 -6822.157} C_VEL
LIN {X 0,Y 481.741,Z 274.786,A -85,B 0,C 180,E1 -6824.775,E2 -6824.775} C_VEL
LIN {X 0,Y 481.752,Z 274.779,A -85,B 0,C 180,E1 -6828.215,E2 -6828.215} C_VEL
LIN {X 0,Y 481.739,Z 274.792,A -85,B 0,C 180,E1 -6831.611,E2 -6831.611} C_VEL
LIN {X 0,Y 481.809,Z 274.77,A -85,B 0,C 180,E1 -6834.139,E2 -6834.139} C_VEL
LIN {X 0,Y 481.919,Z 274.771,A -85,B 0,C 180,E1 -6837.492,E2 -6837.492} C_VEL
LIN {X 0,Y 481.941,Z 274.753,A -85,B 0,C 180,E1 -6840,E2 -6840} C_VEL
LIN {X 0,Y 481.927,Z 274.762,A -85,B 0,C 180,E1 -6842.507,E2 -6842.507} C_VEL
LIN {X 0,Y 481.8,Z 274.772,A -85,B 0,C 180,E1 -6845.86,E2 -6845.86} C_VEL
LIN {X 0,Y 481.763,Z 274.777,A -85,B 0,C 180,E1 -6848.388,E2 -6848.388} C_VEL
LIN {X 0,Y 481.751,Z 274.784,A -85,B 0,C 180,E1 -6851.784,E2 -6851.784} C_VEL
LIN {X 0,Y 481.742,Z 274.792,A -85,B 0,C 180,E1 -6855.224,E2 -6855.224} C_VEL
LIN {X 0,Y 481.708,Z 274.793,A -85,B 0,C 180,E1 -6858.721,E2 -6858.721} C_VEL
LIN {X 0,Y 481.645,Z 274.802,A -85,B 0,C 180,E1 -6861.394,E2 -6861.394} C_VEL
LIN {X 0,Y 481.677,Z 274.795,A -85,B 0,C 180,E1 -6864.113,E2 -6864.113} C_VEL
LIN {X 0,Y 481.746,Z 274.792,A -85,B 0,C 180,E1 -6867.139,E2 -6867.139} C_VEL
LIN {X 0,Y 481.678,Z 274.795,A -85,B 0,C 180,E1 -6869.741,E2 -6869.741} C_VEL
LIN {X 0,Y 481.671,Z 274.799,A -85,B 0,C 180,E1 -6872.674,E2 -6872.674} C_VEL
LIN {X 0,Y 481.64,Z 274.796,A -85,B 0,C 180,E1 -6875.709,E2 -6875.709} C_VEL
LIN {X 0,Y 481.671,Z 274.802,A -85,B 0,C 180,E1 -6878.859,E2 -6878.859} C_VEL
LIN {X 0,Y 481.661,Z 274.797,A -85,B 0,C 180,E1 -6881.914,E2 -6881.914} C_VEL
LIN {X 0,Y 481.659,Z 274.797,A -85,B 0,C 180,E1 -6884.457,E2 -6884.457} C_VEL
LIN {X 0,Y 481.652,Z 274.796,A -85,B 0,C 180,E1 -6887.84,E2 -6887.84} C_VEL
LIN {X 0,Y 481.679,Z 274.8,A -85,B 0,C 180,E1 -6890.651,E2 -6890.651} C_VEL
LIN {X 0,Y 481.625,Z 274.803,A -85,B 0,C 180,E1 -6893.376,E2 -6893.376} C_VEL
LIN {X 0,Y 481.708,Z 274.791,A -85,B 0,C 180,E1 -6896.33,E2 -6896.33} C_VEL
LIN {X 0,Y 481.681,Z 274.961,A -85,B 0,C 180,E1 -6897.712,E2 -6897.712} C_VEL
LIN {X 0,Y 488.269,Z 296.602,A -85,B 0,C 180,E1 -6900.451,E2 -6900.451} C_VEL
LIN {X 0,Y 489.074,Z 300.715,A -85,B 0,C 180,E1 -6900.931,E2 -6900.931} C_VEL
LIN {X 0,Y 488.567,Z 310.05,A -85,B 0,C 180,E1 -6901.858,E2 -6901.858} C_VEL
LIN {X 0,Y 492.574,Z 333.227,A -85,B 0,C 180,E1 -6902.466,E2 -6902.466} C_VEL
LIN {X 0,Y 490.309,Z 515.062,A -85,B 0,C 180,E1 -6905.249,E2 -6905.249} C_VEL
LIN {X 0,Y 489.774,Z 531.474,A -85,B 0,C 180,E1 -6905.635,E2 -6905.635} C_VEL
LIN {X 0,Y 489.158,Z 547.243,A -85,B 0,C 180,E1 -6906.166,E2 -6906.166} C_VEL
LIN {X 0,Y 488.314,Z 562.9,A -85,B 0,C 180,E1 -6906.853,E2 -6906.853} C_VEL
LIN {X 0,Y 487.429,Z 578.544,A -85,B 0,C 180,E1 -6907.732,E2 -6907.732} C_VEL
LIN {X 0,Y 486.468,Z 591.509,A -85,B 0,C 180,E1 -6908.606,E2 -6908.606} C_VEL
LIN {X 0,Y 485.582,Z 604.911,A -85,B 0,C 180,E1 -6909.674,E2 -6909.674} C_VEL
LIN {X 0,Y 484.556,Z 618.44,A -85,B 0,C 180,E1 -6910.953,E2 -6910.953} C_VEL
LIN {X 0,Y 483.732,Z 629.941,A -85,B 0,C 180,E1 -6912.236,E2 -6912.236} C_VEL
LIN {X 0,Y 482.963,Z 641.63,A -85,B 0,C 180,E1 -6913.754,E2 -6913.754} C_VEL
LIN {X 0,Y 482.325,Z 651.377,A -85,B 0,C 180,E1 -6915.227,E2 -6915.227} C_VEL
LIN {X 0,Y 481.803,Z 660.896,A -85,B 0,C 180,E1 -6916.933,E2 -6916.933} C_VEL
LIN {X 0,Y 481.428,Z 668.865,A -85,B 0,C 180,E1 -6918.634,E2 -6918.634} C_VEL
LIN {X 0,Y 481.075,Z 675.513,A -85,B 0,C 180,E1 -6920.328,E2 -6920.328} C_VEL
LIN {X 0,Y 480.984,Z 680.909,A -85,B 0,C 180,E1 -6922.021,E2 -6922.021} C_VEL
LIN {X 0,Y 480.91,Z 684.91,A -85,B 0,C 180,E1 -6923.587,E2 -6923.587} C_VEL
LIN {X 0,Y 480.832,Z 687.665,A -85,B 0,C 180,E1 -6924.969,E2 -6924.969} C_VEL
LIN {X 0,Y 480.867,Z 690.154,A -85,B 0,C 180,E1 -6926.649,E2 -6926.649} C_VEL
LIN {X 0,Y 480.784,Z 691.555,A -85,B 0,C 180,E1 -6928.325,E2 -6928.325} C_VEL
LIN {X 0,Y 480.738,Z 692.08,A -85,B 0,C 180,E1 -6930,E2 -6930} C_VEL
LIN {X 0,Y 480.813,Z 691.548,A -85,B 0,C 180,E1 -6931.675,E2 -6931.675} C_VEL
LIN {X 0,Y 480.867,Z 690.14,A -85,B 0,C 180,E1 -6933.352,E2 -6933.352} C_VEL
LIN {X 0,Y 480.832,Z 687.646,A -85,B 0,C 180,E1 -6935.031,E2 -6935.031} C_VEL
LIN {X 0,Y 480.904,Z 684.219,A -85,B 0,C 180,E1 -6936.714,E2 -6936.714} C_VEL
LIN {X 0,Y 481.03,Z 678.354,A -85,B 0,C 180,E1 -6938.825,E2 -6938.825} C_VEL
LIN {X 0,Y 481.324,Z 670.643,A -85,B 0,C 180,E1 -6940.942,E2 -6940.942} C_VEL
LIN {X 0,Y 481.715,Z 662.966,A -85,B 0,C 180,E1 -6942.641,E2 -6942.641} C_VEL
LIN {X 0,Y 482.147,Z 653.797,A -85,B 0,C 180,E1 -6944.347,E2 -6944.347} C_VEL
LIN {X 0,Y 482.77,Z 644.392,A -85,B 0,C 180,E1 -6945.84,E2 -6945.84} C_VEL
LIN {X 0,Y 483.498,Z 633.388,A -85,B 0,C 180,E1 -6947.337,E2 -6947.337} C_VEL
LIN {X 0,Y 484.306,Z 622.345,A -85,B 0,C 180,E1 -6948.618,E2 -6948.618} C_VEL
LIN {X 0,Y 485.296,Z 608.381,A -85,B 0,C 180,E1 -6950.008,E2 -6950.008} C_VEL
LIN {X 0,Y 486.315,Z 594.361,A -85,B 0,C 180,E1 -6951.179,E2 -6951.179} C_VEL
LIN {X 0,Y 487.308,Z 579.921,A -85,B 0,C 180,E1 -6952.191,E2 -6952.191} C_VEL
LIN {X 0,Y 488.31,Z 564.103,A -85,B 0,C 180,E1 -6953.091,E2 -6953.091} C_VEL
LIN {X 0,Y 489.117,Z 548.934,A -85,B 0,C 180,E1 -6953.78,E2 -6953.78} C_VEL
LIN {X 0,Y 489.808,Z 532.207,A -85,B 0,C 180,E1 -6954.363,E2 -6954.363} C_VEL
LIN {X 0,Y 490.408,Z 516.366,A -85,B 0,C 180,E1 -6954.749,E2 -6954.749} C_VEL
LIN {X 0,Y 492.822,Z 333.136,A -85,B 0,C 180,E1 -6957.588,E2 -6957.588} C_VEL
LIN {X 0,Y 488.719,Z 309.595,A -85,B 0,C 180,E1 -6958.242,E2 -6958.242} C_VEL
LIN {X 0,Y 489.296,Z 299.995,A -85,B 0,C 180,E1 -6959.233,E2 -6959.233} C_VEL
LIN {X 0,Y 485.176,Z 285.696,A -85,B 0,C 180,E1 -6961.086,E2 -6961.086} C_VEL
LIN {X 0,Y 481.66,Z 274.799,A -85,B 0,C 180,E1 -6962.605,E2 -6962.605} C_VEL
LIN {X 0,Y 481.661,Z 274.8,A -85,B 0,C 180,E1 -6965.205,E2 -6965.205} C_VEL
LIN {X 0,Y 481.671,Z 274.797,A -85,B 0,C 180,E1 -6968.859,E2 -6968.859} C_VEL
LIN {X 0,Y 481.662,Z 274.792,A -85,B 0,C 180,E1 -6971.915,E2 -6971.915} C_VEL
LIN {X 0,Y 481.66,Z 274.798,A -85,B 0,C 180,E1 -6974.458,E2 -6974.458} C_VEL
LIN {X 0,Y 481.648,Z 274.795,A -85,B 0,C 180,E1 -6977.84,E2 -6977.84} C_VEL
LIN {X 0,Y 481.681,Z 274.798,A -85,B 0,C 180,E1 -6980.651,E2 -6980.651} C_VEL
LIN {X 0,Y 481.627,Z 274.802,A -85,B 0,C 180,E1 -6983.377,E2 -6983.377} C_VEL
LIN {X 0,Y 481.71,Z 274.789,A -85,B 0,C 180,E1 -6986.33,E2 -6986.33} C_VEL
LIN {X 0,Y 481.651,Z 274.799,A -85,B 0,C 180,E1 -6989.418,E2 -6989.418} C_VEL
LIN {X 0,Y 481.7,Z 274.78,A -85,B 0,C 180,E1 -6992.169,E2 -6992.169} C_VEL
LIN {X 0,Y 481.72,Z 274.792,A -85,B 0,C 180,E1 -6994.97,E2 -6994.97} C_VEL
LIN {X 0,Y 481.651,Z 274.787,A -85,B 0,C 180,E1 -6997.705,E2 -6997.705} C_VEL
LIN {X 0,Y 481.706,Z 274.794,A -85,B 0,C 180,E1 -7000.394,E2 -7000.394} C_VEL
LIN {X 0,Y 481.688,Z 274.783,A -85,B 0,C 180,E1 -7003.034,E2 -7003.034} C_VEL
LIN {X 0,Y 481.688,Z 274.792,A -85,B 0,C 180,E1 -7005.639,E2 -7005.639} C_VEL
LIN {X 0,Y 481.753,Z 274.783,A -85,B 0,C 180,E1 -7008.216,E2 -7008.216} C_VEL
LIN {X 0,Y 481.738,Z 274.785,A -85,B 0,C 180,E1 -7011.612,E2 -7011.612} C_VEL
LIN {X 0,Y 481.791,Z 274.781,A -85,B 0,C 180,E1 -7014.14,E2 -7014.14} C_VEL
LIN {X 0,Y 481.922,Z 274.761,A -85,B 0,C 180,E1 -7017.493,E2 -7017.493} C_VEL
LIN {X 0,Y 481.94,Z 274.764,A -85,B 0,C 180,E1 -7020,E2 -7020} C_VEL
LIN {X 0,Y 481.912,Z 274.757,A -85,B 0,C 180,E1 -7022.508,E2 -7022.508} C_VEL
LIN {X 0,Y 481.788,Z 274.783,A -85,B 0,C 180,E1 -7025.861,E2 -7025.861} C_VEL
LIN {X 0,Y 481.723,Z 274.78,A -85,B 0,C 180,E1 -7028.389,E2 -7028.389} C_VEL
LIN {X 0,Y 481.754,Z 274.787,A -85,B 0,C 180,E1 -7031.785,E2 -7031.785} C_VEL
LIN {X 0,Y 481.733,Z 274.784,A -85,B 0,C 180,E1 -7035.225,E2 -7035.225} C_VEL
LIN {X 0,Y 481.707,Z 274.78,A -85,B 0,C 180,E1 -7038.722,E2 -7038.722} C_VEL
LIN {X 0,Y 481.645,Z 274.799,A -85,B 0,C 180,E1 -7041.395,E2 -7041.395} C_VEL
LIN {X 0,Y 481.645,Z 274.794,A -85,B 0,C 180,E1 -7044.115,E2 -7044.115} C_VEL
LIN {X 0,Y 481.644,Z 274.797,A -85,B 0,C 180,E1 -7047.115,E2 -7047.115} C_VEL
LIN {X 0,Y 481.603,Z 274.805,A -85,B 0,C 180,E1 -7049.747,E2 -7049.747} C_VEL
LIN {X 0,Y 481.636,Z 274.801,A -85,B 0,C 180,E1 -7052.678,E2 -7052.678} C_VEL
LIN {X 0,Y 481.64,Z 274.799,A -85,B 0,C 180,E1 -7055.2,E2 -7055.2} C_VEL
LIN {X 0,Y 481.623,Z 274.803,A -85,B 0,C 180,E1 -7058.002,E2 -7058.002} C_VEL
LIN {X 0,Y 481.606,Z 274.803,A -85,B 0,C 180,E1 -7061.048,E2 -7061.048} C_VEL
LIN {X 0,Y 481.653,Z 274.801,A -85,B 0,C 180,E1 -7064.459,E2 -7064.459} C_VEL
LIN {X 0,Y 481.632,Z 274.849,A -85,B 0,C 180,E1 -7066.969,E2 -7066.969} C_VEL
LIN {X 0,Y 484.925,Z 285.673,A -85,B 0,C 180,E1 -7068.552,E2 -7068.552} C_VEL
LIN {X 0,Y 492.435,Z 301.542,A -85,B 0,C 180,E1 -7069.322,E2 -7069.322} C_VEL
LIN {X 0,Y 493.063,Z 305.488,A -85,B 0,C 180,E1 -7069.428,E2 -7069.428} C_VEL
LIN {X 0,Y 491.596,Z 412.712,A -85,B 0,C 180,E1 -7071.084,E2 -7071.084} C_VEL
LIN {X 0,Y 490.95,Z 418.565,A -85,B 0,C 180,E1 -7071.14,E2 -7071.14} C_VEL
LIN {X 0,Y 485.535,Z 437.662,A -85,B 0,C 180,E1 -7071.123,E2 -7071.123} C_VEL
LIN {X 0,Y 484.879,Z 443.516,A -85,B 0,C 180,E1 -7071.179,E2 -7071.179} C_VEL
LIN {X 0,Y 484.184,Z 491.642,A -85,B 0,C 180,E1 -7071.951,E2 -7071.951} C_VEL
LIN {X 0,Y 483.56,Z 508.765,A -85,B 0,C 180,E1 -7072.396,E2 -7072.396} C_VEL
LIN {X 0,Y 482.872,Z 524.655,A -85,B 0,C 180,E1 -7072.986,E2 -7072.986} C_VEL
LIN {X 0,Y 481.963,Z 540.361,A -85,B 0,C 180,E1 -7073.737,E2 -7073.737} C_VEL
LIN {X 0,Y 481.084,Z 554.585,A -85,B 0,C 180,E1 -7074.583,E2 -7074.583} C_VEL
LIN {X 0,Y 479.994,Z 569.807,A -85,B 0,C 180,E1 -7075.687,E2 -7075.687} C_VEL
LIN {X 0,Y 478.922,Z 583.374,A -85,B 0,C 180,E1 -7076.874,E2 -7076.874} C_VEL
LIN {X 0,Y 477.872,Z 596.29,A -85,B 0,C 180,E1 -7078.209,E2 -7078.209} C_VEL
LIN {X 0,Y 476.887,Z 608.41,A -85,B 0,C 180,E1 -7079.685,E2 -7079.685} C_VEL
LIN {X 0,Y 476.119,Z 618.334,A -85,B 0,C 180,E1 -7081.091,E2 -7081.091} C_VEL
LIN {X 0,Y 475.398,Z 628.102,A -85,B 0,C 180,E1 -7082.723,E2 -7082.723} C_VEL
LIN {X 0,Y 474.945,Z 635.31,A -85,B 0,C 180,E1 -7084.118,E2 -7084.118} C_VEL
LIN {X 0,Y 474.449,Z 643.375,A -85,B 0,C 180,E1 -7085.961,E2 -7085.961} C_VEL
LIN {X 0,Y 474.105,Z 649.857,A -85,B 0,C 180,E1 -7087.79,E2 -7087.79} C_VEL
LIN {X 0,Y 473.944,Z 655.022,A -85,B 0,C 180,E1 -7089.606,E2 -7089.606} C_VEL
LIN {X 0,Y 473.708,Z 659.536,A -85,B 0,C 180,E1 -7091.718,E2 -7091.718} C_VEL
LIN {X 0,Y 473.603,Z 662.314,A -85,B 0,C 180,E1 -7093.623,E2 -7093.623} C_VEL
LIN {X 0,Y 473.607,Z 663.726,A -85,B 0,C 180,E1 -7095.388,E2 -7095.388} C_VEL
LIN {X 0,Y 473.651,Z 664.203,A -85,B 0,C 180,E1 -7097.14,E2 -7097.14} C_VEL
LIN {X 0,Y 473.716,Z 663.616,A -85,B 0,C 180,E1 -7098.88,E2 -7098.88} C_VEL
LIN {X 0,Y 473.631,Z 662.12,A -85,B 0,C 180,E1 -7100.606,E2 -7100.606} C_VEL
LIN {X 0,Y 473.735,Z 659.585,A -85,B 0,C 180,E1 -7102.327,E2 -7102.327} C_VEL
LIN {X 0,Y 473.916,Z 656.075,A -85,B 0,C 180,E1 -7104.041,E2 -7104.041} C_VEL
LIN {X 0,Y 474.051,Z 651.521,A -85,B 0,C 180,E1 -7105.749,E2 -7105.749} C_VEL
LIN {X 0,Y 474.216,Z 645.861,A -85,B 0,C 180,E1 -7107.452,E2 -7107.452} C_VEL
LIN {X 0,Y 474.668,Z 639.046,A -85,B 0,C 180,E1 -7109.152,E2 -7109.152} C_VEL
LIN {X 0,Y 475.165,Z 629.748,A -85,B 0,C 180,E1 -7111.059,E2 -7111.059} C_VEL
LIN {X 0,Y 475.925,Z 619.787,A -85,B 0,C 180,E1 -7112.751,E2 -7112.751} C_VEL
LIN {X 0,Y 476.792,Z 609.557,A -85,B 0,C 180,E1 -7114.226,E2 -7114.226} C_VEL
LIN {X 0,Y 477.718,Z 597.657,A -85,B 0,C 180,E1 -7115.699,E2 -7115.699} C_VEL
LIN {X 0,Y 478.703,Z 584.683,A -85,B 0,C 180,E1 -7117.063,E2 -7117.063} C_VEL
LIN {X 0,Y 479.784,Z 570.406,A -85,B 0,C 180,E1 -7118.317,E2 -7118.317} C_VEL
LIN {X 0,Y 480.674,Z 557.629,A -85,B 0,C 180,E1 -7119.255,E2 -7119.255} C_VEL
LIN {X 0,Y 481.656,Z 542.41,A -85,B 0,C 180,E1 -7120.19,E2 -7120.19} C_VEL
LIN {X 0,Y 482.439,Z 527.928,A -85,B 0,C 180,E1 -7120.916,E2 -7120.916} C_VEL
LIN {X 0,Y 483.256,Z 511.036,A -85,B 0,C 180,E1 -7121.562,E2 -7121.562} C_VEL
LIN {X 0,Y 483.818,Z 495.009,A -85,B 0,C 180,E1 -7122,E2 -7122} C_VEL
LIN {X 0,Y 484.206,Z 472.928,A -85,B 0,C 180,E1 -7122.389,E2 -7122.389} C_VEL
LIN {X 0,Y 486.383,Z 305.657,A -85,B 0,C 180,E1 -7124.97,E2 -7124.97} C_VEL
LIN {X 0,Y 484.707,Z 301.132,A -85,B 0,C 180,E1 -7125.144,E2 -7125.144} C_VEL
LIN {X 0,Y 477.466,Z 285.382,A -85,B 0,C 180,E1 -7125.857,E2 -7125.857} C_VEL
LIN {X 0,Y 474.636,Z 275.674,A -85,B 0,C 180,E1 -7127.254,E2 -7127.254} C_VEL
LIN {X 0,Y 474.652,Z 275.674,A -85,B 0,C 180,E1 -7129.91,E2 -7129.91} C_VEL
LIN {X 0,Y 474.638,Z 275.675,A -85,B 0,C 180,E1 -7133.358,E2 -7133.358} C_VEL
LIN {X 0,Y 474.575,Z 275.677,A -85,B 0,C 180,E1 -7136.377,E2 -7136.377} C_VEL
LIN {X 0,Y 474.598,Z 275.678,A -85,B 0,C 180,E1 -7139.253,E2 -7139.253} C_VEL
LIN {X 0,Y 474.589,Z 275.682,A -85,B 0,C 180,E1 -7142.424,E2 -7142.424} C_VEL
LIN {X 0,Y 474.591,Z 275.675,A -85,B 0,C 180,E1 -7145.464,E2 -7145.464} C_VEL
LIN {X 0,Y 474.581,Z 275.679,A -85,B 0,C 180,E1 -7148.46,E2 -7148.46} C_VEL
LIN {X 0,Y 474.582,Z 275.679,A -85,B 0,C 180,E1 -7151.79,E2 -7151.79} C_VEL
LIN {X 0,Y 474.615,Z 275.674,A -85,B 0,C 180,E1 -7155.298,E2 -7155.298} C_VEL
LIN {X 0,Y 474.582,Z 275.682,A -85,B 0,C 180,E1 -7158.21,E2 -7158.21} C_VEL
LIN {X 0,Y 474.587,Z 275.672,A -85,B 0,C 180,E1 -7161.54,E2 -7161.54} C_VEL
LIN {X 0,Y 474.611,Z 275.661,A -85,B 0,C 180,E1 -7164.724,E2 -7164.724} C_VEL
LIN {X 0,Y 474.627,Z 275.678,A -85,B 0,C 180,E1 -7167.786,E2 -7167.786} C_VEL
LIN {X 0,Y 474.599,Z 275.668,A -85,B 0,C 180,E1 -7170.89,E2 -7170.89} C_VEL
LIN {X 0,Y 474.584,Z 275.684,A -85,B 0,C 180,E1 -7173.623,E2 -7173.623} C_VEL
LIN {X 0,Y 474.636,Z 275.664,A -85,B 0,C 180,E1 -7176.642,E2 -7176.642} C_VEL
LIN {X 0,Y 474.655,Z 275.669,A -85,B 0,C 180,E1 -7180.089,E2 -7180.089} C_VEL
LIN {X 0,Y 474.635,Z 275.665,A -85,B 0,C 180,E1 -7182.773,E2 -7182.773} C_VEL
LIN {X 0,Y 474.643,Z 275.676,A -85,B 0,C 180,E1 -7185.42,E2 -7185.42} C_VEL
LIN {X 0,Y 474.706,Z 275.657,A -85,B 0,C 180,E1 -7188.037,E2 -7188.037} C_VEL
LIN {X 0,Y 474.711,Z 275.669,A -85,B 0,C 180,E1 -7191.486,E2 -7191.486} C_VEL
LIN {X 0,Y 474.772,Z 275.647,A -85,B 0,C 180,E1 -7194.052,E2 -7194.052} C_VEL
LIN {X 0,Y 474.884,Z 275.647,A -85,B 0,C 180,E1 -7197.455,E2 -7197.455} C_VEL
LIN {X 0,Y 474.912,Z 275.629,A -85,B 0,C 180,E1 -7200,E2 -7200} C_VEL
LIN {X 0,Y 474.893,Z 275.638,A -85,B 0,C 180,E1 -7202.544,E2 -7202.544} C_VEL
LIN {X 0,Y 474.761,Z 275.648,A -85,B 0,C 180,E1 -7205.947,E2 -7205.947} C_VEL
LIN {X 0,Y 474.728,Z 275.654,A -85,B 0,C 180,E1 -7208.513,E2 -7208.513} C_VEL
LIN {X 0,Y 474.705,Z 275.661,A -85,B 0,C 180,E1 -7211.962,E2 -7211.962} C_VEL
LIN {X 0,Y 474.699,Z 275.667,A -85,B 0,C 180,E1 -7215.455,E2 -7215.455} C_VEL
LIN {X 0,Y 474.662,Z 275.673,A -85,B 0,C 180,E1 -7219.01,E2 -7219.01} C_VEL
LIN {X 0,Y 474.588,Z 275.677,A -85,B 0,C 180,E1 -7221.728,E2 -7221.728} C_VEL
LIN {X 0,Y 474.659,Z 275.671,A -85,B 0,C 180,E1 -7224.492,E2 -7224.492} C_VEL
LIN {X 0,Y 474.68,Z 275.669,A -85,B 0,C 180,E1 -7227.334,E2 -7227.334} C_VEL
LIN {X 0,Y 474.604,Z 275.676,A -85,B 0,C 180,E1 -7230.23,E2 -7230.23} C_VEL
LIN {X 0,Y 474.642,Z 275.675,A -85,B 0,C 180,E1 -7233.22,E2 -7233.22} C_VEL
LIN {X 0,Y 474.591,Z 275.674,A -85,B 0,C 180,E1 -7236.323,E2 -7236.323} C_VEL
LIN {X 0,Y 474.626,Z 275.672,A -85,B 0,C 180,E1 -7239.647,E2 -7239.647} C_VEL
LIN {X 0,Y 474.639,Z 275.678,A -85,B 0,C 180,E1 -7242.931,E2 -7242.931} C_VEL
LIN {X 0,Y 474.613,Z 275.676,A -85,B 0,C 180,E1 -7245.896,E2 -7245.896} C_VEL
LIN {X 0,Y 474.631,Z 275.677,A -85,B 0,C 180,E1 -7249.04,E2 -7249.04} C_VEL
LIN {X 0,Y 474.608,Z 275.675,A -85,B 0,C 180,E1 -7251.704,E2 -7251.704} C_VEL
LIN {X 0,Y 474.622,Z 275.674,A -85,B 0,C 180,E1 -7254.726,E2 -7254.726} C_VEL
LIN {X 0,Y 474.645,Z 275.747,A -85,B 0,C 180,E1 -7257.322,E2 -7257.322} C_VEL
LIN {X 0,Y 480.828,Z 296.092,A -85,B 0,C 180,E1 -7259.945,E2 -7259.945} C_VEL
LIN {X 0,Y 482.419,Z 302.576,A -85,B 0,C 180,E1 -7260.735,E2 -7260.735} C_VEL
LIN {X 0,Y 481.998,Z 309.968,A -85,B 0,C 180,E1 -7261.464,E2 -7261.464} C_VEL
LIN {X 0,Y 486.219,Z 334.32,A -85,B 0,C 180,E1 -7262.113,E2 -7262.113} C_VEL
LIN {X 0,Y 483.779,Z 515.906,A -85,B 0,C 180,E1 -7264.926,E2 -7264.926} C_VEL
LIN {X 0,Y 483.243,Z 531.751,A -85,B 0,C 180,E1 -7265.313,E2 -7265.313} C_VEL
LIN {X 0,Y 482.569,Z 548.053,A -85,B 0,C 180,E1 -7265.877,E2 -7265.877} C_VEL
LIN {X 0,Y 481.656,Z 563.511,A -85,B 0,C 180,E1 -7266.571,E2 -7266.571} C_VEL
LIN {X 0,Y 480.74,Z 578.554,A -85,B 0,C 180,E1 -7267.429,E2 -7267.429} C_VEL
LIN {X 0,Y 479.67,Z 592.622,A -85,B 0,C 180,E1 -7268.4,E2 -7268.4} C_VEL
LIN {X 0,Y 478.719,Z 605.923,A -85,B 0,C 180,E1 -7269.493,E2 -7269.493} C_VEL
LIN {X 0,Y 477.672,Z 619.227,A -85,B 0,C 180,E1 -7270.78,E2 -7270.78} C_VEL
LIN {X 0,Y 476.744,Z 631.498,A -85,B 0,C 180,E1 -7272.188,E2 -7272.188} C_VEL
LIN {X 0,Y 475.908,Z 642.825,A -85,B 0,C 180,E1 -7273.716,E2 -7273.716} C_VEL
LIN {X 0,Y 475.271,Z 652.408,A -85,B 0,C 180,E1 -7275.222,E2 -7275.222} C_VEL
LIN {X 0,Y 474.717,Z 661.791,A -85,B 0,C 180,E1 -7276.952,E2 -7276.952} C_VEL
LIN {X 0,Y 474.268,Z 670.479,A -85,B 0,C 180,E1 -7278.893,E2 -7278.893} C_VEL
LIN {X 0,Y 473.953,Z 678.178,A -85,B 0,C 180,E1 -7281.043,E2 -7281.043} C_VEL
LIN {X 0,Y 473.822,Z 684.034,A -85,B 0,C 180,E1 -7283.185,E2 -7283.185} C_VEL
LIN {X 0,Y 473.758,Z 687.459,A -85,B 0,C 180,E1 -7284.894,E2 -7284.894} C_VEL
LIN {X 0,Y 473.773,Z 689.948,A -85,B 0,C 180,E1 -7286.598,E2 -7286.598} C_VEL
LIN {X 0,Y 473.689,Z 691.348,A -85,B 0,C 180,E1 -7288.3,E2 -7288.3} C_VEL
LIN {X 0,Y 473.664,Z 691.873,A -85,B 0,C 180,E1 -7290,E2 -7290} C_VEL
LIN {X 0,Y 473.715,Z 691.34,A -85,B 0,C 180,E1 -7291.7,E2 -7291.7} C_VEL
LIN {X 0,Y 473.773,Z 689.931,A -85,B 0,C 180,E1 -7293.402,E2 -7293.402} C_VEL
LIN {X 0,Y 473.759,Z 687.435,A -85,B 0,C 180,E1 -7295.107,E2 -7295.107} C_VEL
LIN {X 0,Y 473.822,Z 684.006,A -85,B 0,C 180,E1 -7296.815,E2 -7296.815} C_VEL
LIN {X 0,Y 473.953,Z 678.138,A -85,B 0,C 180,E1 -7298.957,E2 -7298.957} C_VEL
LIN {X 0,Y 474.268,Z 670.424,A -85,B 0,C 180,E1 -7301.107,E2 -7301.107} C_VEL
LIN {X 0,Y 474.658,Z 662.743,A -85,B 0,C 180,E1 -7302.832,E2 -7302.832} C_VEL
LIN {X 0,Y 475.152,Z 653.578,A -85,B 0,C 180,E1 -7304.563,E2 -7304.563} C_VEL
LIN {X 0,Y 475.834,Z 643.827,A -85,B 0,C 180,E1 -7306.129,E2 -7306.129} C_VEL
LIN {X 0,Y 476.613,Z 633.191,A -85,B 0,C 180,E1 -7307.595,E2 -7307.595} C_VEL
LIN {X 0,Y 477.46,Z 622.167,A -85,B 0,C 180,E1 -7308.895,E2 -7308.895} C_VEL
LIN {X 0,Y 478.505,Z 608.596,A -85,B 0,C 180,E1 -7310.27,E2 -7310.27} C_VEL
LIN {X 0,Y 479.539,Z 595.685,A -85,B 0,C 180,E1 -7311.381,E2 -7311.381} C_VEL
LIN {X 0,Y 480.61,Z 581.157,A -85,B 0,C 180,E1 -7312.425,E2 -7312.425} C_VEL
LIN {X 0,Y 481.633,Z 566.082,A -85,B 0,C 180,E1 -7313.317,E2 -7313.317} C_VEL
LIN {X 0,Y 482.535,Z 550.317,A -85,B 0,C 180,E1 -7314.068,E2 -7314.068} C_VEL
LIN {X 0,Y 483.299,Z 534.274,A -85,B 0,C 180,E1 -7314.656,E2 -7314.656} C_VEL
LIN {X 0,Y 483.976,Z 518.317,A -85,B 0,C 180,E1 -7315.069,E2 -7315.069} C_VEL
LIN {X 0,Y 484.571,Z 477.96,A -85,B 0,C 180,E1 -7315.728,E2 -7315.728} C_VEL
LIN {X 0,Y 486.599,Z 334.272,A -85,B 0,C 180,E1 -7317.972,E2 -7317.972} C_VEL
LIN {X 0,Y 482.673,Z 311.541,A -85,B 0,C 180,E1 -7318.617,E2 -7318.617} C_VEL
LIN {X 0,Y 482.271,Z 309.136,A -85,B 0,C 180,E1 -7318.706,E2 -7318.706} C_VEL
LIN {X 0,Y 482.651,Z 301.86,A -85,B 0,C 180,E1 -7319.476,E2 -7319.476} C_VEL
LIN {X 0,Y 478.523,Z 287.657,A -85,B 0,C 180,E1 -7321.357,E2 -7321.357} C_VEL
LIN {X 0,Y 474.637,Z 275.673,A -85,B 0,C 180,E1 -7323.064,E2 -7323.064} C_VEL
LIN {X 0,Y 474.588,Z 275.68,A -85,B 0,C 180,E1 -7326.324,E2 -7326.324} C_VEL
LIN {X 0,Y 474.627,Z 275.675,A -85,B 0,C 180,E1 -7329.648,E2 -7329.648} C_VEL
LIN {X 0,Y 474.635,Z 275.673,A -85,B 0,C 180,E1 -7332.932,E2 -7332.932} C_VEL
LIN {X 0,Y 474.609,Z 275.674,A -85,B 0,C 180,E1 -7335.896,E2 -7335.896} C_VEL
LIN {X 0,Y 474.628,Z 275.67,A -85,B 0,C 180,E1 -7339.041,E2 -7339.041} C_VEL
LIN {X 0,Y 474.61,Z 275.671,A -85,B 0,C 180,E1 -7341.704,E2 -7341.704} C_VEL
LIN {X 0,Y 474.624,Z 275.678,A -85,B 0,C 180,E1 -7344.726,E2 -7344.726} C_VEL
LIN {X 0,Y 474.636,Z 275.667,A -85,B 0,C 180,E1 -7347.788,E2 -7347.788} C_VEL
LIN {X 0,Y 474.624,Z 275.668,A -85,B 0,C 180,E1 -7350.885,E2 -7350.885} C_VEL
